// TIA Portal V19 export
FUNCTION_BLOCK "LAF_ProfinetDevDiag"   // FB73, LAD
TITLE = LAF_ProfinetDevDiag / Profinet Device Diagnose mit ProDiag
AUTHOR : Siemens Digital Industries
FAMILY : LAF
VERSION : 1.2
// The block is used for the diagnostics of the Profinet devices connected to a CPU and to display the information on the HMI. The following data will be read from the PLC and displayed via faceplates.
// * Device state 
// * Device name (max. 24 characters) 
// * Device number 
// * Group status of module errors 
// * first 8 characters of the order number (MLFB) 
// 
// The function block has to be called and configured; and the faceplates for each device have to be placed in a screen and supplied with the interface.  
// 
//  
// **PLC Data types**  
// * LAF_typeDevDiagAlarm  
// * LAF_typeDevDiagBasic  
// * LAF_typeDevDiagGlobal  
// * LAF_typeDevDiagHwAddress  
// * LAF_typeDevDiagInstruct  
// * LAF_typeDevDiagInterface  
// * LAF_typeDevDiagInternal  
// * LAF_typeDevDiagModStateMode  
// * LAF_typeDevDiagNoOfDevices  
// * LAF_typeDevDiagRisEdge  
// * LAF_typeDevDiagState  
// * LAF_typeDevDiagStateInstruct  
// * LAF_typeDevDiagStatesMode  
// * LAF_typeDevDiagStructGetDiag  
// 
// **User Constants**  
// MAX_NO_OF_MODULES  
// MAX_NO_OF_DEVICES  
// 
// 
// **WinCC Screen**  
// ![Image](LAF_ProfinetDevDiag_PrD/en/image1.PNG)
// 
// **Block call example**  
// {.pageWidth}
// ![Image]( LAF_ProfinetDevDiag_PrD/en/image42.PNG)  
// 
// **Calling interface**  
// The block must be called only once per PROFINET-IO-System in the cyclic program. The call takes place in the software unit CentralFunctions -> [CallDiagnostic](../Functions/CallDiagnostic.htm)  
// 
// **Internally used „Extended instructions / blocks“**  
// LOG2GEO, DeviceStates, GEO2LOG, ModuleStates, Get_Name, GET_IM_DATA, GET_DIAG  
// 
// **Parameters**  
// This block is provided with “pre-defined actual parameters” for structured data types, user constants, system constants etc. Therefor these parameters have to be modified only slightly or not at all, if the symbols of DBs, user constants, and system constants have not been changed.
// Die Tec-Unit diagnostiziert die an die CPU angeschlossenen Profinet Geräte um die Informationen auf dem HMI darzustellen. Folgend Daten werden gelesen und mittels eines Bildbausteins visualisiert.  
// * Geräte-Status 
// * Gerätename (max. 24 Zeichen) 
// * Geräte-Nummer 
// * Sammelzustand über Modulstörung 
// * die ersten 8 Zeichen der Bestell-/Artikelnummer (MLFB) 
// 
// Hierzu muss der Funktionsbaustein aufgerufen und parametriert werden, sowie für jedes Profinet-Gerät der vorgefertigte Bildbaustein (Faceplate) in einem Bild platziert, und mit der Schnittstelle versorgt werden.  
//  
//  
// **PLC-Datentypen**  
// 
// ![Image](LSicar_ProfinetDevDiag_PrD/de/image3.PNG)
//  
// 
// **Anwenderkonstanten**  
// MAX_NO_OF_MODULES  
// MAX_NO_OF_DEVICES  
// 
// **WinCC-Bildbaustein**  
// 
// ![Image](LSicar_ProfinetDevDiag_PrD/de/image1.PNG)
// 
// **WinCC-Bild**  
// 
// ![Image](LSicar_ProfinetDevDiag_PrD/de/image2.PNG)
// 
// **Beispielaufruf**  
// Abbildung in Kontaktplan (KOP), ohne Parameterbeschaltung. D:\Software\Symbols_Icons\BMPs-JPGs-PNGs\Verschiedene\symb_user_goto_transparent.pngEin lauffähiger Programm-Aufruf hierzu ist im „SICAR-StartUp“-Projekt enthalten.  
// 
// **Aufrufschnittstelle**  
// Der Baustein wird einmalig pro PROFINET-IO-System im zyklischen Programm aufgerufen.  
// 
// **Intern verwendete „Erweiterte Anweisungen / Bausteine“**  
// LOG2GEO, DeviceStates, GEO2LOG, ModuleStates, Get_Name, GET_IM_DATA, GET_DIAG  
// 
// **Parameter**  
// 
// ![Icon](_Icon/information.PNG)
// 
// Der Baustein ist mit "Vordefinierten Aktualparametern" versehen für Strukturvariablen, Anwender- und Systemkonstanten etc., die dadurch nicht oder nur geringfügig angepasst werden müssen, vorausgesetzt die Symbolischen Namen von DBs, Anwender-/Systemkonstanten etc. wurden nicht geändert. Die Anpassungen sind notwendig beim Index [i], z.B. für den BA-Bereich oder die HMI-/Panelnummer.  
// * Der Index ist vorbesetzt mit dem Wert [0]. Damit wird auf den Index 0 (Dummy) verwiesen. Sofern der Baustein-Parameter nicht benötigt wird, sind keine Anpassungen notwendig, andernfalls muss der Indexwert angepasst werden. 
// oder  
// * Der Index ist vorbesetzt mit [???]. Dies führt dazu, dass der Aktualparameter beim Bausteinaufruf rot markiert wird; um darauf aufmerksam zu machen, dass der Indexwert des Aktualparameters angepasst werden muss!
// stored: Access Published, IsIECCheckEnabled true, MemoryReserve 100, SetENOAutomatically true
   VAR_INPUT
      plantIdentifier { ExternalAccessible := 'False'; ExternalVisible := 'False'; ExternalWritable := 'False'} : WString[#MAX_CHAR];   // Betriebsmittel Kennzeichen. Das Kennzeichen ist auf 24 Zeichen begrenzt und sollte ein Be-triebsmittelkennzeichen, gemäß der Schaltpläne enthalten. Der Text wird im Bildbaustein, und in der Bewegungszeile ange-zeigt bzw. als Präfix für die Alarme benutzt / Identifier of the device. The identifier is limited to a length of 24 characters and should contain the name of the device according the wiring diagrams. The identifier is displayed in the faceplate and it is used as a prefix for the alarm messages.
      textListId { ExternalAccessible := 'False'; ExternalVisible := 'False'; ExternalWritable := 'False'} : Int;   // Text list ID
      localProfinetSystem { ExternalAccessible := 'False'; ExternalVisible := 'False'; ExternalWritable := 'False'} : HW_IOSYSTEM;   // Systemkonstante des lokalen „Profinet IO-Systems“. Die Variab-le befindet sich in den PLC-Variablen unter „Alle Variablen anzei-gen -> Lasche Systemkonstanten“. / System constant of the local Profinet IO system. The tag is located in PLC tags / Show all tags ->tab “System constants”.
      firstCycle { ExternalAccessible := 'False'; ExternalVisible := 'False'; ExternalWritable := 'False'} : Bool;   // Variable die den ersten CPU-Zyklus darstellt. Der Parameter ist vordefiniert und verweist auf nachfolgende Quelle. / Tag representing the first PLC cycle.
      maxDevicesDiag { ExternalAccessible := 'False'; ExternalVisible := 'False'; ExternalWritable := 'False'} : DInt;   // Maximale Anzahl von PN Devices. Der Parameter ist vordefiniert und verweist auf nachfolgende Quelle. / Maximum number of PN devices.
      maxModulesDiag { ExternalAccessible := 'False'; ExternalVisible := 'False'; ExternalWritable := 'False'} : DInt;   // Maximale Anzahl von Modulen „Der Parameter ist vordefiniert und verweist auf nachfolgende Quelle. / Maximum number of modules.
      ackAlarms { ExternalAccessible := 'False'; ExternalVisible := 'False'; ExternalWritable := 'False'} : Bool;   // Variable für Alarm quittieren. Es wird empfohlen die Variable “GlobalInterface”.globalHmi.globalAck zu verwenden. Die Varibriable wird durch den Quittier Button in der Kopfzeile versorgt. / Tag for Reset of alarms. It is recommended to use the tag “GlobalInterface”.globalHmi.globalAck” representing the Acknowledge “ACK” button in the screen header.
      hideAlarmAll { ExternalAccessible := 'False'; ExternalVisible := 'False'; ExternalWritable := 'False'} : Bool;   // Alle Störungen unterdrücken. Mit Signal TRUE werden alle Alarme unterdrückt. Hinweis: Die farbliche Animation des WinCC-Bildbausteins im PN-Diagnosebild wird immer ausgeführt. / Hide all alarms. Signal TRUE on this input, will suppress all alarms. Note: The WinCC-Faceplate in the PN-Screen will be always animated.
      hideAlarmMask { ExternalAccessible := 'False'; ExternalVisible := 'False'; ExternalWritable := 'False'} : Word;   // Einzelne Störungen unterdrücken. Bei Bedarf können einzelne Alarme deaktiviert werden, durch Setzen des entsprechenden Bits auf TRUE. Hinweis: Die farbliche Animation des WinCC-Bildbausteins im PN-Diagnosebild wird immer ausgeführt. / Hide alarm mask. Individual alarms can be suppressed by setting the corresponding bit in this mask to state TRUE (This might be necessary e.g. during commissioning). The assignment is the same as in tag “statAlarm”.
   END_VAR
   VAR_OUTPUT
      generalAlarm { ExternalAccessible := 'False'; ExternalVisible := 'False'; ExternalWritable := 'False'} : Bool;   // Sammelstörung / Group alarm.
      deviceFaulty { ExternalAccessible := 'False'; ExternalVisible := 'False'; ExternalWritable := 'False'} : Bool;   // TRUE = mindestens 1 Profinet Gerät gestört ist. / TRUE = at least one device in condition fault.
      deviceProblem { ExternalAccessible := 'False'; ExternalVisible := 'False'; ExternalWritable := 'False'} : Bool;   // TRUE = mindestens 1 Profinet Gerät ein Problem aufweist. / TRUE = at least one device with a problem.
      deviceDeactivated { ExternalAccessible := 'False'; ExternalVisible := 'False'; ExternalWritable := 'False'} : Bool;   // TRUE = mindestens 1 Profinet Gerät deaktiviert ist. / TRUE = at least one device deactivated.
      deviceNotPresent { ExternalAccessible := 'False'; ExternalVisible := 'False'; ExternalWritable := 'False'} : Bool;   // mind. 1 PN-Device nicht vorhanden, jedoch konfiguriert (z.B. ausgeschaltet) / Min. 1 device not present, but configured (e.g. switched off ).
   END_VAR
   VAR_IN_OUT
      interfaceDevDiag : "LAF_typeDevDiagInterface";   // This parameter refers to the data block "InstDevDiagInterface", which contains the information for the HMI as well as a user interface about the status of the devices. / Dieser Parameter verweist auf den Datenbaustein "DevDiagInterface“, der die Informationen für das HMI sowie eine Anwender-Schnittstelle über den Status der Devices enthält.
   END_VAR
   VAR
      statDevDiagInternal { ExternalAccessible := 'False'; ExternalVisible := 'False'; ExternalWritable := 'False'} : "LAF_typeDevDiagInternal";   // für HMI (Erreichbarkeit setzen) / for HMI (set accessebility)
      statCnt1ShotGetName { ExternalAccessible := 'False'; ExternalVisible := 'False'; ExternalWritable := 'False'} : DInt := 1;   // Einmalig "GetName": Zykluszähler PN-Devices, läuft von 1...PN_DEVDIAG_MAX-DEVICES, beginnt dann wieder bei 1 / Once only "GetName" cycle counter
      statCnt1ShotGeo2Log { ExternalAccessible := 'False'; ExternalVisible := 'False'; ExternalWritable := 'False'} : DInt := 1;   // Einmalig "GEO2LOG": Zykluszähler PN-Devices, läuft von 1...PN_DEVDIAG_MAX-DEVICES, beginnt dann wieder bei 1 / Once only "GEO2LOG" cycle counter
      statCnt1ShotGetImDat { ExternalAccessible := 'False'; ExternalVisible := 'False'; ExternalWritable := 'False'} : DInt := 1;   // Einmalig "GET_IM_DATA": Zykluszähler PN-Devices, läuft von 1...PN_DEVDIAG_MAX-DEVICES, beginnt dann wieder bei 1 / Once only "GET_IM_DATA" cycle counter
      statCntCyclDevState { ExternalAccessible := 'False'; ExternalVisible := 'False'; ExternalWritable := 'False'} : DInt := 1;   // Zyklisch für "DeviceStates": Zykluszähler PN-Devices, läuft von 1...5, beginnt dann wieder bei 1 / Cyclic "DeviceStates"cycle counter
      statCntCyclState { ExternalAccessible := 'False'; ExternalVisible := 'False'; ExternalWritable := 'False'} : DInt := 1;   // Zyklisch für "DeviceStates" rangieren in Device-Arrays: Zykluszähler PN-Devices, läuft von 1...5, beginnt dann wieder bei 1 / Cyclic "DeviceStates" cycle counter, routing to device-arrays
      statCntCyclModulState { ExternalAccessible := 'False'; ExternalVisible := 'False'; ExternalWritable := 'False'} : DInt := 1;   // Zyklisch für "ModuleStates": Zykluszähler PN-Devices, läuft von 1...PN_DEVDIAG_MAX-DEVICES, beginnt dann wieder bei 1 / Cyclic "ModuleStates" cycle counter
      statCntCyclGetDiag { ExternalAccessible := 'False'; ExternalVisible := 'False'; ExternalWritable := 'False'} : DInt := 1;   // Zyklisch für "GET_DIAG": Zykluszähler PN-Devices, läuft von 1...PN_DEVDIAG_MAX-DEVICES, beginnt dann wieder bei 1 / Cyclic "GET_DIAG" cycle counter
      statBusy { ExternalAccessible := 'False'; ExternalVisible := 'False'; ExternalWritable := 'False'} : "LAF_typeDevDiagStateInstruct";   // Busy_flags
      statDone { ExternalAccessible := 'False'; ExternalVisible := 'False'; ExternalWritable := 'False'} : "LAF_typeDevDiagStateInstruct";   // Done_flags
      statOtherInstruct { ExternalAccessible := 'False'; ExternalVisible := 'False'; ExternalWritable := 'False'} : "LAF_typeDevDiagInstruct";   // Instanzen fuer Instructions
      instGetName { ExternalAccessible := 'False'; ExternalVisible := 'False'; ExternalWritable := 'False'} : Get_Name;   // Instanzen Get_Name / Instance Get_Name
      statGetNameDat { ExternalAccessible := 'False'; ExternalVisible := 'False'; ExternalWritable := 'False'} : String[#LENGTH_GET_NAME];   // Get_Name: Name der Baugruppe / Get_Name: Name of device
      statGetNameErrorStatus { ExternalAccessible := 'False'; ExternalVisible := 'False'; ExternalWritable := 'False'} : Word;   // Get name error status
      statGetNameErrorDevCycle { ExternalAccessible := 'False'; ExternalVisible := 'False'; ExternalWritable := 'False'} : DInt;   // Zykluszähler für PN-Devices, läuft von 1...PN_DEVDIAG_MAX-DEVICES und beginnt dann wieder bei 1 usw. / Cyclic counter PN devices 1..MAX_DEVICES
      instGetImData { ExternalAccessible := 'False'; ExternalVisible := 'False'; ExternalWritable := 'False'} : Get_IM_Data;   // GET_IM_DATA
      statIm0Data { ExternalAccessible := 'False'; ExternalVisible := 'False'; ExternalWritable := 'False'} : IM0_Data;   // GET_IM_DATA
      statGetImDatErrorStatus { ExternalAccessible := 'False'; ExternalVisible := 'False'; ExternalWritable := 'False'} : Word;   // Get IM data error status
      statGetImDatErrorCycle { ExternalAccessible := 'False'; ExternalVisible := 'False'; ExternalWritable := 'False'} : DInt;   // Zykluszähler für PN-Devices, läuft von 1...PN_DEVDIAG_MAX-DEVICES und beginnt dann wieder bei 1 usw. / Cyclic counter PN devices 1..MAX_DEVICES
      statAlarm { ExternalAccessible := 'False'; ExternalVisible := 'False'; ExternalWritable := 'False'} : "LAF_typeDevDiagAlarm";   // Störungen / Alarm
      statHideAlarm { ExternalAccessible := 'False'; ExternalVisible := 'False'; ExternalWritable := 'False'} : "LAF_typeDevDiagAlarm";   // Störungen unterdrücken, Belegung identisch mit "Alarm" / Hide Alarms, identical with "Alarm"
      statRisPushbutton { ExternalAccessible := 'False'; ExternalVisible := 'False'; ExternalWritable := 'False'} : "LAF_typeDevDiagRisEdge";   // Flankenauswertung Tasten / Edge evaluation buttons
      statErrorText { ExternalAccessible := 'False'; ExternalVisible := 'False'; ExternalWritable := 'False'} : String[#LENGTH_GET_NAME] := 'No Device Name readable';   // Error text / Fehlertext
      stat8CharError { ExternalAccessible := 'False'; ExternalVisible := 'False'; ExternalWritable := 'False'} : String[#LENGTH_8_CHAR] := '????????';   // 8 character error / 8 Zeichen Fehler
      statAlarmNo { ExternalAccessible := 'False'; ExternalVisible := 'False'; ExternalWritable := 'False'} : Array[0..23] of UInt;   // Alarm Nummer für ProDiag / Alarm Number for ProDiag
   END_VAR
   VAR_TEMP
      tempDevCnt1ShotGetName : UInt;   // Type conversion / Typ Konvertierung
      tempHideAlarm : Word;   // Abbild hideAlarmMask / Image hideAlarmMask
      tempZeroWord : Word;   // Word Konstante=0 / Word constant=0
      tempZeroDword : DWord;   // DWord Konstante=0 / DWord constant=0
      tempAlarmStatus : Word;   // Abbild statAlarm / image statAlarm
   END_VAR
   VAR CONSTANT
      MAX_CHAR : DInt := 24;   // Konstante für Zeichenlänge plantidentifier / Constant length plantidentifier
      LENGTH_GET_NAME : DInt := 24;   // Length GetName / Zeichenlänge GetName
      LENGTH_8_CHAR : DInt := 8;   // Constant 8 character / Länge 8 Zeichen
   END_VAR
   // statAlarmNo[0] := 0;
   // statAlarmNo[1] := 1;
   // statAlarmNo[2] := 2;
   // statAlarmNo[3] := 3;
   // statAlarmNo[4] := 4;
   // statAlarmNo[5] := 5;
   // statAlarmNo[6] := 6;
   // statAlarmNo[7] := 7;
   // statAlarmNo[8] := 8;
   // statAlarmNo[9] := 9;
   // statAlarmNo[10] := 10;
   // statAlarmNo[11] := 11;
   // statAlarmNo[12] := 12;
   // statAlarmNo[13] := 13;
   // statAlarmNo[14] := 14;
   // statAlarmNo[15] := 15;
   // statAlarmNo[16] := 16;
   // statAlarmNo[17] := 17;
   // statAlarmNo[18] := 18;
   // statAlarmNo[19] := 19;
   // statAlarmNo[20] := 20;
   // statAlarmNo[21] := 21;
   // statAlarmNo[22] := 22;
   // statAlarmNo[23] := 23;
   VAR_TEMP   // added for the SCL form of the ladder/FBD networks
      _w1 : Bool;
      _w2 : Bool;
      _w3 : Bool;
      _w4 : Bool;
   END_VAR
BEGIN

REGION Network 1: Header Info / Änderungshistorie
   // SIEMENS AG / (c)Copyright 2024
   // ------------------------------------------------------------------------------
   // Title:            LAF_InterfaceSignalsBool
   // Comment/Function: The block is used for the diagnostics of the Profinet devices connected to a CPU and to display the information on the HMI. 
   // Library/Family:   Library of Automation Framework
   // Author:               Siemens Digital Industry
   // Tested with:      S7-PLCSIM Advanced 6.0
   // Engineering:     TIA Portal V19
   // Restrictions:      --- 
   // Requirements:  ---
   // ------------------------------------------------------------------------------
   // Change log table:
   // Version | Date | Expert in charge | Changes applied
   // -------|---------|-------------|--------------------------------------------
   // 01.02.00 | 30.09.2024 | SIMATIC Systems Support | First released version
   // Die Änderungshistorie wird nur in englischer Editiersprache geführt.
END_REGION

REGION Network 2: Description / Beschreibung
   // **Operation mode Automatic / Manual**  
   // The block is not assigned to any operation mode.  
   // 
   // **Alarms**  
   // Alarm texts are stored in the PLC alarm text lists of the software unit GlobalData. This messages are used with proDiag and also in the program alarm version of the block.  
   // 
   // | **No.** | **Message**                                                            |
   // |---------|------------------------------------------------------------------------|
   // | 1       | Invalid Value / Userconstant   "PNDevDiag": MAX_NO_OF_DEVICES [1..]     |
   // | 2       | Invalid Value / Userconstant "PNDevDiag": MAX_NO_OF_MODULES   [1..128] |
   // | 3       | Invalid Address "PNDevDiag": LOG2GEO_LOCAL_PNIO-SYSTEM                 |
   // | 4       | PROFINET Device-States: Error Read Device-States                       |
   // | 5       | PROFINET-Device faulty                                                 |
   // | 6       | PROFINET-Device with Problem                                           |
   // | 7       | Spare7                                                                 |
   // | 8       | PROFINET-Device not present but configured                             |
   // | 9       | PROFINET-Device with network error (e.g. Topology-error)               |
   // | 10      | POFINET-Device with maintenance required                               |
   // | 11      | POFINET-Device with maintenance demanded                               |
   // | 12      | Spare12                                                                |
   // | 13      | Spare13                                                                |
   // | 14      | Spare14                                                                |
   // | 15      | Spare15                                                                |
   // | 16      | Spare16                                                                |
   // | 17      | Spare17                                                                |
   // | 18      | Hide all alarm active                                                  |
   // 
   // ---
   // 
   // **User Constants**  
   // User constants are available under  the SW unit “CentralFunctions -> PLC tags -> 11_Settings -> User constants”  
   // 
   // {.pageWidth}
   // ![Image](LAF_ProfinetDevDiag_PrD/en/image4.PNG)
   // 
   // **MAX_NO_OF_DEVICES**  
   // The value of the constant should be adapted to the real number of used devices.  
   // 
   // **MAX_NO_OF_MODULES**  
   // The value of the constant should be adapted to the maximum number of used modules in a I/O station.  
   // 
   // NOTE
   // :     These values have impact on the update time of data and cycle time.  
   // 
   // ---
   // 
   // 
   // #### PLC Data types 
   // * [LAF_typeDevDiagAlarm](../Library%20Types/LAF_typeDevDiagAlarm.htm)  
   // * [LAF_typeDevDiagBasic](../Library%20Types/LAF_typeDevDiagBasic.htm)  
   // * [LAF_typeDevDiagGlobal](../Library%20Types/LAF_typeDevDiagGlobal.htm)  
   // * [LAF_typeDevDiagHwAddress](../Library%20Types/LAF_typeDevDiagHwAddress.htm)  
   // * [LAF_typeDevDiagInstruct](../Library%20Types/LAF_typeDevDiagInstruct.htm)  
   // * [LAF_typeDevDiagInterface](../Library%20Types/LAF_typeDevDiagInterface.htm)  
   // * [LAF_typeDevDiagInternal](../Library%20Types/LAF_typeDevDiagInternal.htm)  
   // * [LAF_typeDevDiagModStateMode](../Library%20Types/LAF_typeDevDiagModStateMode.htm)  
   // * [LAF_typeDevDiagNoOfDevices](../Library%20Types/LAF_typeDevDiagNoOfDevices.htm)  
   // * [LAF_typeDevDiagRisEdge](../Library%20Types/LAF_typeDevDiagRisEdge.htm)  
   // * [LAF_typeDevDiagState](../Library%20Types/LAF_typeDevDiagState.htm)  
   // * [LAF_typeDevDiagStateInstruct](../Library%20Types/LAF_typeDevDiagStateInstruct.htm)  
   // * [LAF_typeDevDiagStatesMode](../Library%20Types/LAF_typeDevDiagStatesMode.htm)  
   // * [LAF_typeDevDiagStructGetDiag](../Library%20Types/LAF_typeDevDiagStructGetDiag.htm)  
   // 
   // #### InstDevDiagInterface DB 
   // The data block “PNDevDiagInterface“is derived from the data type „LAF_typeDevDiagInterface“ and contains all information for the status to display on HMI as well as a user interface to evaluate the status program internally.  
   // {.pageWidth}
   // ![Image](LAF_ProfinetDevDiag_PrD/en/image19.PNG)
   // 
   // ---
   // 
   // **Global information**  
   // {.pageWidth}
   // ![Image](LAF_ProfinetDevDiag_PrD/en/image20.PNG)
   // 
   // ---
   // 
   // **Device status for display on HMI**  
   // {.pageWidth}
   // ![Image](LAF_ProfinetDevDiag_PrD/en/image21.PNG)
   // 
   // ---
   // 
   // **User interface device status**  
   // {.pageWidth}
   // ![Image](LAF_ProfinetDevDiag_PrD/en/image22.PNG)
   // 
   // ---
   // 
   // #### WinCC-Screen objects 
   // 
   // **WinCC Faceplate**  
   // 
   // The faceplate is available in the project library under Types -> LAF -> 10_Central -> Diagnostic -> ProfinetDevice_Diag.  
   // The faceplate consists of several WinCC objects and contains the information shown below.  
   // The faceplate is animated in terms of color depending on status and operation.   
   // 
   // {.pageWidth}
   // ![Image](LAF_ProfinetDevDiag_PrD/en/image23.PNG)
   // 
   // 
   // **WinCC Faceplate interface connection**  
   // In order to connect the faceplate with the interface tag for a Profinet device it is recommended to proceed as follows:  
   // 
   // 1. For each device, a HMI tag is available.  
   // 2. The faceplate from the project library needs to be placed in the template screen.  
   // 
   // NOTE
   // 
   // :     The data interface is available in data block „InstDevDiagInterface“.  
   // :     The array index number corresponds with the device number.  
   // :     Index [0] are not used.  
   // :     The tag has to be assigned to Properties -> Interface -> HMI.
   // 
   // ---
   // 
   // **WinCC Screen template for placement of the faceplates**  
   // The faceplate is available in the project navigation under Screens -> 09_Diagnostics -> 53_PnDiagnostic.  
   // The screen consists of several WinCC objects and contains the shown below information.  
   // 
   // {.pageWidth}
   // ![Image](LAF_ProfinetDevDiag_PrD/en/image40.PNG)
   // 
   // 
   // #### Further information 
   // 
   // #### Update info 
   //  
   // #### Further documentation
   // **Betriebsart Automatik / Hand**  
   // Der Baustein ist keiner Betriebsart / Betriebsartenbereich zugeordnet.  
   // 
   // **Alarme**  
   // Anstehende Alarme können über die OUTPUT-Parameter für den weiteren Programmablauf verwendet werden.  Alarme können über den „QUIT“-Button im HMI-Bild quittiert werden.  
   // 
   // **Alarm**  
   // Die statische Strukturvariable „statAlarm“ hat folgende Belegung:  
   // 
   // |       statAlarm. [Word]  |  |  |
   // |---|---|---|
   // |     Bitposition  |   Bezeichnung  |   Erläuterung  |
   // |     %X0  |   #.invalidValueMaxDevices  |   Input kleiner/gleich angegeben, muss grösser/gleich 1 sein [1..]  |
   // |     %X1  |   #.invalidValueMaxModules  |   Input kleiner/gleich 0 oder grösser angegeben, gültig [1..128]  |
   // |     %X2  |   #.InvalidAddressLog2Geo  |   ungültige Adresse an LADDR bei LOG2GEO bzw. an Input  |
   // |     %X3  |   #.errorReadDeviceState  |   Fehler beim Lesen der Baugruppenzustandsinformationen  |
   // |     %X4  |   #.deviceFaulty  |   mind. 1 PN-Device gestört  |
   // |     %X5  |   #.deviceProblem  |   mind. 1 PN-Device hat ein Problem  |
   // |     %X6  |   #.deviceDeactivated  |   mind. 1 PN-Device deaktiviert -Dies ist kein Fehler, lediglich in Struktur gelistet-  |
   // |     %X7  |   #.deviceNotPresent  |   mind. 1 PN-Device nicht vorhanden, jedoch konfiguriert (z.B. konfiguriert und ausgeschaltet)  |
   // |     %X8  |   #.deviceNetworkError  |   mind. 1 PN-Device mit Netzwerkfehler (z.B. Topologie-Fehler)  |
   // |     %X9  |   #.deviceMaintRequired  |   mind. 1 PN-Device mit Wartungsbedarf  |
   // |     %X10  |   #.deviceMaintDemanded  |   mind. 1 PN-Device mit Wartungsanforderung  |
   // |     %X11 .. 15  |   #.spare..  |   Reserve  |
   // 
   // 
   // **Anwenderkonstanten**  
   // Anwenderkonstanten verfügbar unter PLC-Variablen/Alle Variablen anzeigen -> Anwenderkonstanten.  
   // 
   // {.pageWidth}
   // ![Image](LSicar_ProfinetDevDiag_PrD/de/image4.PNG)
   // 
   // **MAX_NO_OF_DEVICES**  
   // Die Anwenderkonstante sollte, auf die auf die tatsächlichen Anzahl Geräte angepasst werden.  
   // 
   // **MAX_NO_OF_MODULES**  
   // Die Anwenderkonstante sollte, auf die auf die maximale Anzahl Module angepasst werden.  
   // 
   // NOTE
   // :     In Abhängigkeit von dem Wert der Variablen hängt die Aktualisierungszeit der Daten und auch somit auch die Zykluszeit.
   // 
   // ---
   // 
   // #### PLC-Datentypen
   // 
   // Verwendete PLC-Datentypen für den SPS-Programmbaustein / WinCC-Bildbaustein/Faceplate:  
   // 
   // **LSicar_typeDevDiagAlarm**  
   // Dieser PLC-Datentyp beinhaltet die Struktur der möglichen Alarme  
   // 
   // {.pageWidth}
   // ![Image](LSicar_ProfinetDevDiag_PrD/de/image5.PNG)
   //  
   // 
   // **_typeDevDiagBasic**  
   // Dieser PLC-Datentyp beinhaltet die Informationen für den Bildbaustein   
   // 
   // {.pageWidth}
   // ![Image](LSicar_ProfinetDevDiag_PrD/de/image6.PNG)
   // 
   // 
   // **_typeDevDiagGlobal**  
   // Dieser PLC-Datentyp beinhaltet globale Daten, für das HMI-Popup.   
   // 
   // {.pageWidth}
   // ![Image](LSicar_ProfinetDevDiag_PrD/de/image7.PNG) 
   // 
   // 
   // **_typeDevDiagHwAddress**  
   // Dieser PLC-Datentyp beinhaltet Informationen der auszuwertenden HW Typen.  
   // 
   // {.pageWidth}
   // ![Image](LSicar_ProfinetDevDiag_PrD/de/image8.PNG) 
   // 
   // **_typeDevDiagInstruct**  
   // Dieser PLC-Datentyp beinhaltet die Struktur der ausgelesen Diagnose Daten  
   // 
   // {.pageWidth}
   // ![Image](LSicar_ProfinetDevDiag_PrD/de/image9.PNG)
   // 
   // **_typeDevDiagInterface**  
   // Dieser PLC-Datentyp bildet die Struktur für den Datenbaustein „DevDiagInterface“.    
   // 
   // {.pageWidth}
   // ![Image](LSicar_ProfinetDevDiag_PrD/de/image10.PNG) 
   // 
   // **_typeDevDiagInternal**  
   // Dieser PLC-Datentyp beinhaltet interne Daten für die Bearbeitung des Funktionsbausteines, die nicht am HMI angezeigt werden.  
   // 
   // {.pageWidth}
   // ![Image](LSicar_ProfinetDevDiag_PrD/de/image11.PNG) 
   // 
   // **_typeDevDiagModStateMode**  
   // Dieser PLC-Datentyp beinhaltet die Struktur der Parameter sowie die Rückgabewerte der Module.  
   // 
   // {.pageWidth}
   // ![Image](LSicar_ProfinetDevDiag_PrD/de/image12.PNG)
   // 
   // **_typeDevDiagNoOfDevices**  
   // Dieser PLC-Datentyp beinhaltet die Anzahl der Geräte, die diesen Status-Informationen entsprechen.  
   // 
   // {.pageWidth}
   // ![Image](LSicar_ProfinetDevDiag_PrD/de/image13.PNG)
   // 
   // **_typeDevDiagRisEdge**
   // Dieser PLC-Datentyp beinhaltet die Struktur für Flanken-Auswertungen  
   // 
   // {.pageWidth}
   // ![Image](LSicar_ProfinetDevDiag_PrD/de/image14.PNG)
   // 
   // **_typeDevDiagState**  
   // Dieser PLC Datentyp beinhaltet die Status Informationen der Geräte und dient als Anwender-Schnittstelle.   
   // 
   // {.pageWidth}
   // ![Image](LSicar_ProfinetDevDiag_PrD/de/image15.PNG)
   // 
   // **_typeDevDiagStateInstruct**  
   // Dieser PLC-Datentyp beinhaltet die Status Informationen der laufenden Anweisungen.  
   // 
   // {.pageWidth}
   // ![Image](LSicar_ProfinetDevDiag_PrD/de/image16.PNG)
   //  
   // **_typeDevDiagStatesMode**  
   // Dieser PLC-Datentyp beinhaltet die Struktur der Parameter sowie die Rückgabewerte der Geräte.  
   // 
   // {.pageWidth}
   // ![Image](LSicar_ProfinetDevDiag_PrD/de/image17.PNG)
   // 
   // **_typeDevDiagStructGetDiag**  
   // Dieser PLC-Datentyp beinhaltet die Struktur der Anweisung GETDIAG  
   // 
   // {.pageWidth}
   // ![Image](LSicar_ProfinetDevDiag_PrD/de/image18.PNG)
   //  
   // 
   // #### DevDiagInterface DB 
   // Der Datenbaustein „DevDiagInterface“ ist abgeleitet vom PLC Datentyp „LSicar_typeDevDiagInterface“ und beinhaltet sowohl alle Informationen zur Status-Anzeige im HMI als auch eine Anwender-Schnittstelle zur Auswertung des Status für programminterne Zwecke.  
   // 
   // {.pageWidth}
   // ![Image](LSicar_ProfinetDevDiag_PrD/de/image19.PNG)
   // 
   // Global information  
   // 
   // {.pageWidth}
   // ![Image](LSicar_ProfinetDevDiag_PrD/de/image20.PNG)
   // 
   //  
   // Device Status zur Anzeige am HMI  
   // 
   // {.pageWidth}
   // ![Image](LSicar_ProfinetDevDiag_PrD/de/image21.PNG)
   // 
   // Anwender-Schnittstelle Device Status  
   // 
   // {.pageWidth}
   // ![Image](LSicar_ProfinetDevDiag_PrD/de/image22.PNG)
   // 
   // 
   // #### WinCC Bildobjekte 
   // 
   // **WinCC-Bildbaustein**  
   // Der Bildbaustein befindet sich in der Projekt-Bibliothek unter „Typen“.  
   // Der Bildbaustein ist erstellt aus mehreren einzelnen WinCC-Objekten und enthält die dargestellten Informationen. Der Bildbaustein wird farblich animiert, je nach Zustand und Bewegung. Durch Klick auf den Bildbaustein wird in das dazugehörige WinCC (Diagnose) Bild verzweigt, sofern in „Eigenschaften -> Ereignisse“ die entsprechenden Ereignisse projekteirt sind.  
   // 
   // {.pageWidth}
   // ![Image](LSicar_ProfinetDevDiag_PrD/de/image23.PNG)
   // 
   // **Farbgebung / Animation des Bildbausteins (Faceplate)**    
   //  
   //  |       Objekt / Farbe |  |     Bedeutung / Farbe   |
   // |---|---|:---:|
   // |     Profinet Gerätename und Farbanimation  |  |  |
   // |     Gerätename  |   Es wird der in der Hardware-Konfiguration angegeben Gerätename ausgelesen und angezeigt (max. 24 Zeichen).  |  |
   // |     ![Image](LSicar_ProfinetDevDiag_PrD/de/image25.PNG)   |   Gerät ist konfiguriert, vorhanden, aktiviert und fehlerfrei  |  |
   // |     ![Image](LSicar_ProfinetDevDiag_PrD/de/image26.PNG)   |   Gerät ist konfiguriert, aber nicht vorhanden   |  |
   // |     ![Image](LSicar_ProfinetDevDiag_PrD/de/image27.PNG)   |   Gerät ist deaktiviert   |  |
   // |     ![Image](LSicar_ProfinetDevDiag_PrD/de/image28.PNG)   |   Gerät ist gestört   |  |
   // |     ![Image](LSicar_ProfinetDevDiag_PrD/de/image29.PNG)   |   Gerät war gestört   |  |
   // |     ![Image](LSicar_ProfinetDevDiag_PrD/de/image30.PNG)   |   Gerät hat ein Problem   |  |
   // |     ![Image](LSicar_ProfinetDevDiag_PrD/de/image31.PNG)   |   Gerät hatte ein Problem   |  |
   // |     ![Image](LSicar_ProfinetDevDiag_PrD/de/image32.PNG)   |  Kann der Gerätename kann nicht gelesen werden, so wird der Text „No Device Name readable!“ angezeigt. Dies ist ein Hinweis darauf, dass das Gerät möglicherweise nicht konfiguriert und/oder vorhanden ist.   |  |
   // |     Netzsymbol  |  |  |
   // |       ![Image](LSicar_ProfinetDevDiag_PrD/de/image33.PNG)  |  Netzwerk Fehler von Gerät 
   //  - Grün: kein Fehler 
   //  - Rot: Fehler (z.B. Topologiefehler)   |  |
   // |     Gerätenummer  |  |  |
   // |     Beispiel: 25   |   Hier wird die Gerätenummer des Gerätes angezeigt.  |  |
   // |     Modulfehler / Wartung  |  |  |
   // |     ![Image](LSicar_ProfinetDevDiag_PrD/de/image34.PNG)   |   Symbol: Modulfehler  |  |
   // |     ![Image](LSicar_ProfinetDevDiag_PrD/de/image35.PNG)   |   Symbol: Wartungsbedarf  |  |
   // |     ![Image](LSicar_ProfinetDevDiag_PrD/de/image36.PNG)   |   Symbol: Wartungsanforderung  |  |
   // |     Tec-Unit Type  |  |  |
   // |     ![Image](LSicar_ProfinetDevDiag_PrD/de/image37.PNG)   |   Name des Tec-Unit Typs  |  |
   // |     Artikel Bestellnummer (MLFB)  |  |  |
   // |     Beispiel: ![Image](LSicar_ProfinetDevDiag_PrD/de/image38.PNG)   |   Hier werden die ersten 8 Zeichen der Artikel-/Bestellnummer (MLFB) dargestellt. Kann diese Information nicht gelesen werden, so werden ‘????????‘ angezeigt. Dies ist ein Hinweis darauf, dass das Gerät möglicherweise nicht konfiguriert und/oder nicht vorhanden ist.    |  |
   // 
   // 
   // **WinCC-Bildbaustein - Schnittstellenversorgung**  
   // Um den Bildbaustein (Faceplate) für ein Profinet-Gerät mit den notwendigen Daten zu versorgen, gehen Sie wie folgt vor.  
   // 
   // 1. Für jedes PN-Gerät ist eine HMI-Variable angelegt.  
   // 2. Der Bildbaustein aus der Projekt Bibliothek wird in dem Bild platziert. Die Variable muss unter „Eigenschaften -> Schnittstelle“. dem Bildbaustein zugewiesen werden.  
   //   
   // {.pageWidth}
   // ![Image](LSicar_ProfinetDevDiag_PrD/de/image39.PNG)
   // 
   // NOTE
   // :     Die Daten hierzu sind im Datenbaustein „DevDiagInterface“ hinterlegt.  
   // :     Die Index Nummer entspricht der Geräte Nummer. 
   // :     Index [0] wird nicht verwendet. 
   // 
   // ---
   // 
   // **WinCC-Bildvorlage, zur Platzierung der Bildbausteine**  
   // Das Bild befindet sich im Projekt (Projektnavigation) im HMI-Teil unter „Bilder“.  
   // Es ist erstellt aus mehreren einzelnen WinCC-Objekten und enthält die dargestellten Informationen.  
   // 
   // {.pageWidth}
   // ![Image](LSicar_ProfinetDevDiag_PrD/de/image40.PNG)
   // 
   // #### Beispiel 
   // Die Bildbausteine/ Faceplates für die Profinet Geräte Diagnose werden innerhalb eines Bildes platziert und mit der zugehörigen HMI-Variablen verbunden.  
   // Im Beispiel- Bild (rechts) werden die Informationen zur Verfügung gestellt.  
   // 
   // {.pageWidth}
   // ![Image](LSicar_ProfinetDevDiag_PrD/de/image41.PNG)
   // 
   // 
   // #### FWeitere Hinweise
   // 
   // #### Updateinfo 
   //  
   // #### Weitere Dokumente 
   // 
   // ![Icon](_Icon/reference.PNG)
   // 
   // Siehe ..\SICAR_Global\SICAR_Tec-Unit_HMI-Objects.pdf
END_REGION

REGION Network 3: Initialize / Initialisieren
   // Initialization of the values / Initialisieren der Werte
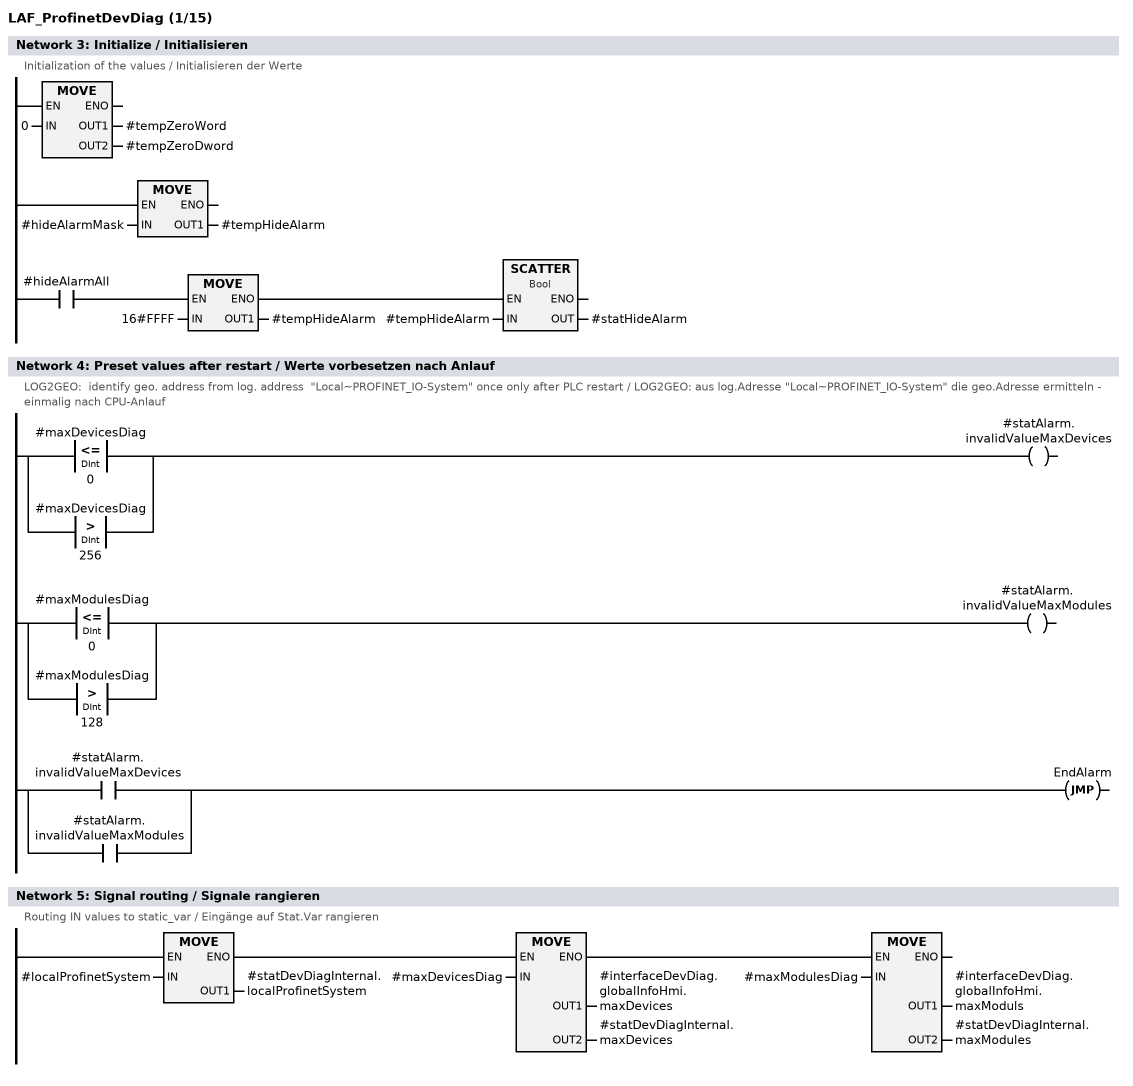
   RUNG wire#powerrail
      Move(in := 0, out1 => #tempZeroWord, out2 => #tempZeroDword)
   END_RUNG
   RUNG wire#powerrail
      Move(in := #hideAlarmMask, out1 => #tempHideAlarm)
   END_RUNG
   RUNG wire#powerrail
      Contact( #hideAlarmAll )
      Move(in := 16#FFFF, out1 => #tempHideAlarm)
      { S7_Templates := "[dest_type := Bool, src_type := Word]" } SCATTER(IN := #tempHideAlarm, OUT => #statHideAlarm)
   END_RUNG
   // the same network as SCL:
   #tempZeroWord := 0;
   #tempZeroDword := 0;
   #tempHideAlarm := #hideAlarmMask;
   IF #hideAlarmAll THEN
       #tempHideAlarm := 16#FFFF;
       SCATTER(IN := #tempHideAlarm, OUT => #statHideAlarm);
   END_IF;
END_REGION

REGION Network 4: Preset values after restart / Werte vorbesetzen nach Anlauf
   // LOG2GEO:  identify geo. address from log. address  "Local~PROFINET_IO-System" once only after PLC restart / LOG2GEO: aus log.Adresse "Local~PROFINET_IO-System" die geo.Adresse ermitteln - einmalig nach CPU-Anlauf
   RUNG wire#powerrail
      { S7_Templates := "SrcType := DInt" } LE_Contact(in1 := #maxDevicesDiag, in2 := 0)
      wire#w1
      Coil( #statAlarm.invalidValueMaxDevices )
   END_RUNG
   RUNG wire#powerrail
      { S7_Templates := "SrcType := DInt" } GT_Contact(in1 := #maxDevicesDiag, in2 := 256)
   END_RUNG wire#w1
   RUNG wire#powerrail
      { S7_Templates := "SrcType := DInt" } LE_Contact(in1 := #maxModulesDiag, in2 := 0)
      wire#w2
      Coil( #statAlarm.invalidValueMaxModules )
   END_RUNG
   RUNG wire#powerrail
      { S7_Templates := "SrcType := DInt" } GT_Contact(in1 := #maxModulesDiag, in2 := 128)
   END_RUNG wire#w2
   RUNG wire#powerrail
      Contact( #statAlarm.invalidValueMaxDevices )
      wire#w3
      JumpCoil( EndAlarm )
   END_RUNG
   RUNG wire#powerrail
      Contact( #statAlarm.invalidValueMaxModules )
   END_RUNG wire#w3
   // the same network as SCL:
   #statAlarm.invalidValueMaxDevices := (#maxDevicesDiag <= 0) OR (#maxDevicesDiag > 256);
   #statAlarm.invalidValueMaxModules := (#maxModulesDiag <= 0) OR (#maxModulesDiag > 128);
   IF #statAlarm.invalidValueMaxDevices OR #statAlarm.invalidValueMaxModules THEN GOTO EndAlarm; END_IF;
END_REGION

REGION Network 5: Signal routing / Signale rangieren
   // Routing IN values to static_var / Eingänge auf Stat.Var rangieren
   RUNG wire#powerrail
      Move(in := #localProfinetSystem, out1 => #statDevDiagInternal.localProfinetSystem)
      Move(in := #maxDevicesDiag, out1 => #interfaceDevDiag.globalInfoHmi.maxDevices, out2 => #statDevDiagInternal.maxDevices)
      Move(in := #maxModulesDiag, out1 => #interfaceDevDiag.globalInfoHmi.maxModuls, out2 => #statDevDiagInternal.maxModules)
   END_RUNG
   // the same network as SCL:
   #statDevDiagInternal.localProfinetSystem := #localProfinetSystem;
   #interfaceDevDiag.globalInfoHmi.maxDevices := #maxDevicesDiag;
   #statDevDiagInternal.maxDevices := #maxDevicesDiag;
   #interfaceDevDiag.globalInfoHmi.maxModuls := #maxModulesDiag;
   #statDevDiagInternal.maxModules := #maxModulesDiag;
END_REGION

REGION Network 6: Initialization / Initialisierung
   // Init after restart PLC or manual request / Initialisierung nach CPU Anlauf
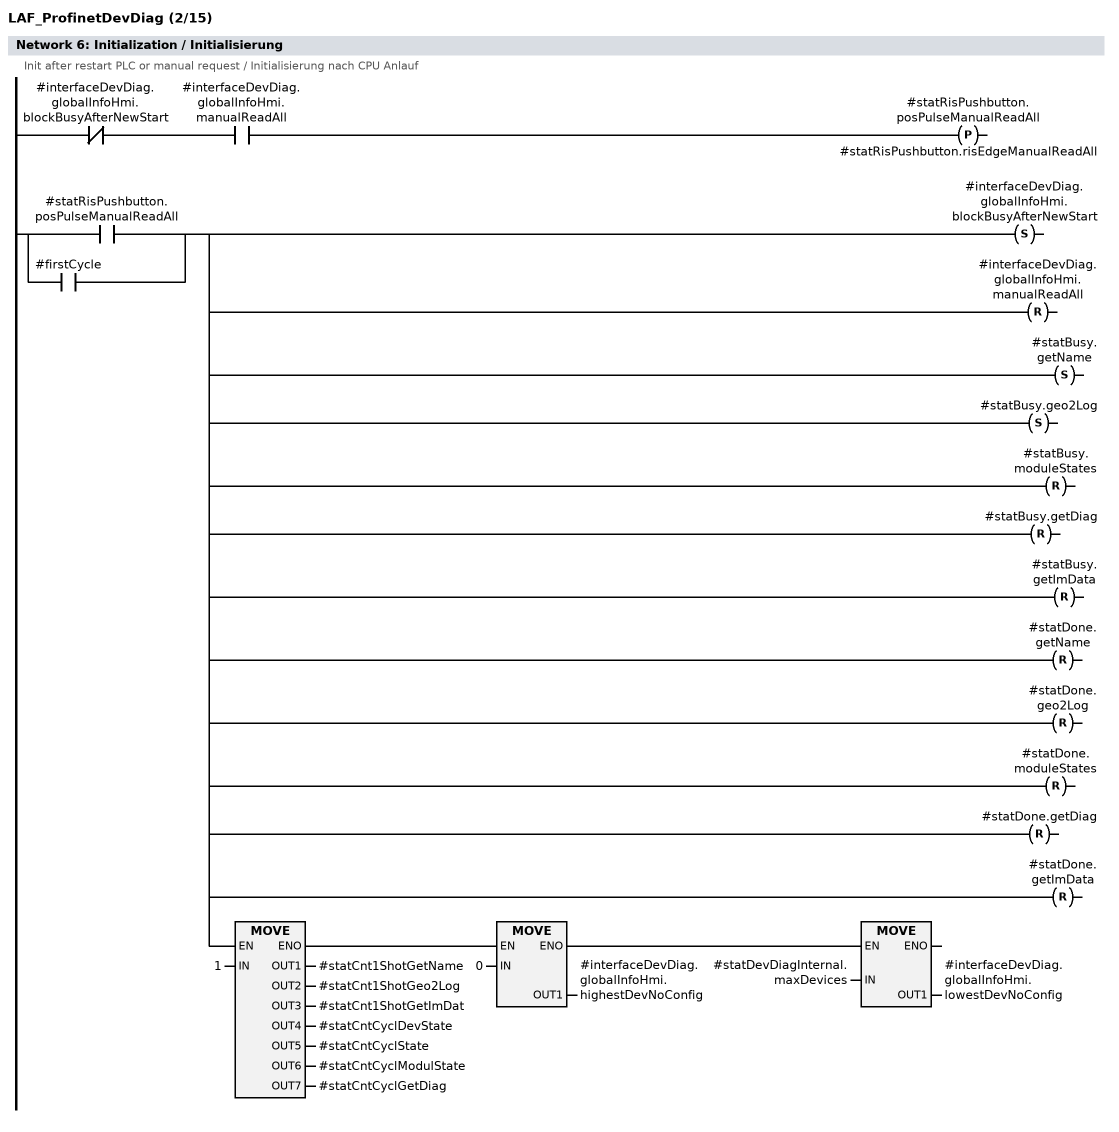
   #_w1 := NOT #interfaceDevDiag.globalInfoHmi.blockBusyAfterNewStart AND #interfaceDevDiag.globalInfoHmi.manualReadAll;
   #statRisPushbutton.posPulseManualReadAll := #_w1 AND NOT #statRisPushbutton.risEdgeManualReadAll;   // rising edge
   #statRisPushbutton.risEdgeManualReadAll := #_w1;
   IF #statRisPushbutton.posPulseManualReadAll OR #firstCycle THEN
       #interfaceDevDiag.globalInfoHmi.blockBusyAfterNewStart := TRUE;
       #interfaceDevDiag.globalInfoHmi.manualReadAll := FALSE;
       #statBusy.getName := TRUE;
       #statBusy.geo2Log := TRUE;
       #statBusy.moduleStates := FALSE;
       #statBusy.getDiag := FALSE;
       #statBusy.getImData := FALSE;
       #statDone.getName := FALSE;
       #statDone.geo2Log := FALSE;
       #statDone.moduleStates := FALSE;
       #statDone.getDiag := FALSE;
       #statDone.getImData := FALSE;
       #statCnt1ShotGetName := 1;
       #statCnt1ShotGeo2Log := 1;
       #statCnt1ShotGetImDat := 1;
       #statCntCyclDevState := 1;
       #statCntCyclState := 1;
       #statCntCyclModulState := 1;
       #statCntCyclGetDiag := 1;
       #interfaceDevDiag.globalInfoHmi.highestDevNoConfig := 0;
       #interfaceDevDiag.globalInfoHmi.lowestDevNoConfig := #statDevDiagInternal.maxDevices;
   END_IF;
END_REGION

REGION Network 7: Read slot number of HW / Lesen der Slotnummer der HW
   // Once only read "LOG2GEO" after restart PLC or manual request, to get the slot number of the HW ID. / Einmailges Lesen LOG2GEO: nach CPU-Neustart oder man. Leseanstoß HMI, um die Slotnummer der HW ID zu erhalten
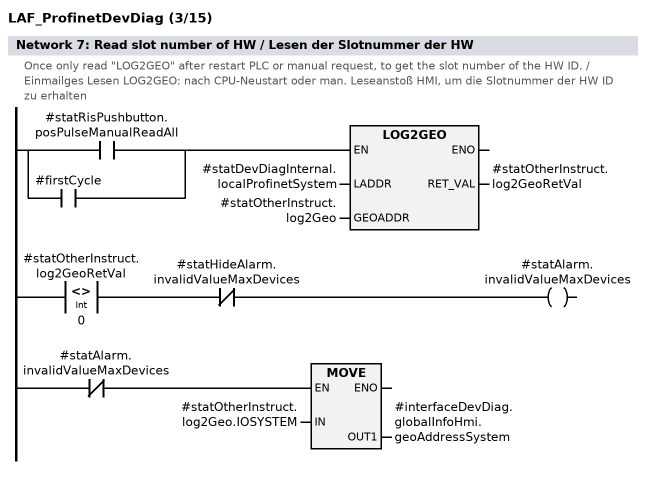
   RUNG wire#powerrail
      Contact( #statRisPushbutton.posPulseManualReadAll )
      wire#w1
      LOG2GEO(LADDR := #statDevDiagInternal.localProfinetSystem, GEOADDR := #statOtherInstruct.log2Geo, Ret_Val => #statOtherInstruct.log2GeoRetVal)
   END_RUNG
   RUNG wire#powerrail
      Contact( #firstCycle )
   END_RUNG wire#w1
   RUNG wire#powerrail
      { S7_Templates := "SrcType := Int" } NE_Contact(in1 := #statOtherInstruct.log2GeoRetVal, in2 := 0)
      I_Contact( #statHideAlarm.invalidValueMaxDevices )
      Coil( #statAlarm.invalidValueMaxDevices )
   END_RUNG
   RUNG wire#powerrail
      I_Contact( #statAlarm.invalidValueMaxDevices )
      Move(in := #statOtherInstruct.log2Geo.IOSYSTEM, out1 => #interfaceDevDiag.globalInfoHmi.geoAddressSystem)
   END_RUNG
   // the same network as SCL:
   IF #statRisPushbutton.posPulseManualReadAll OR #firstCycle THEN
       #statOtherInstruct.log2GeoRetVal := LOG2GEO(LADDR := #statDevDiagInternal.localProfinetSystem,
                               GEOADDR := #statOtherInstruct.log2Geo);
   END_IF;
   #statAlarm.invalidValueMaxDevices := (#statOtherInstruct.log2GeoRetVal <> 0) AND NOT #statHideAlarm.invalidValueMaxDevices;
   IF NOT #statAlarm.invalidValueMaxDevices THEN
       #interfaceDevDiag.globalInfoHmi.geoAddressSystem := #statOtherInstruct.log2Geo.IOSYSTEM;
   END_IF;
END_REGION

REGION Network 8: ResetHistoryAll_HMI
   // Reset of the whole history data / Reseten aller historischer Daten
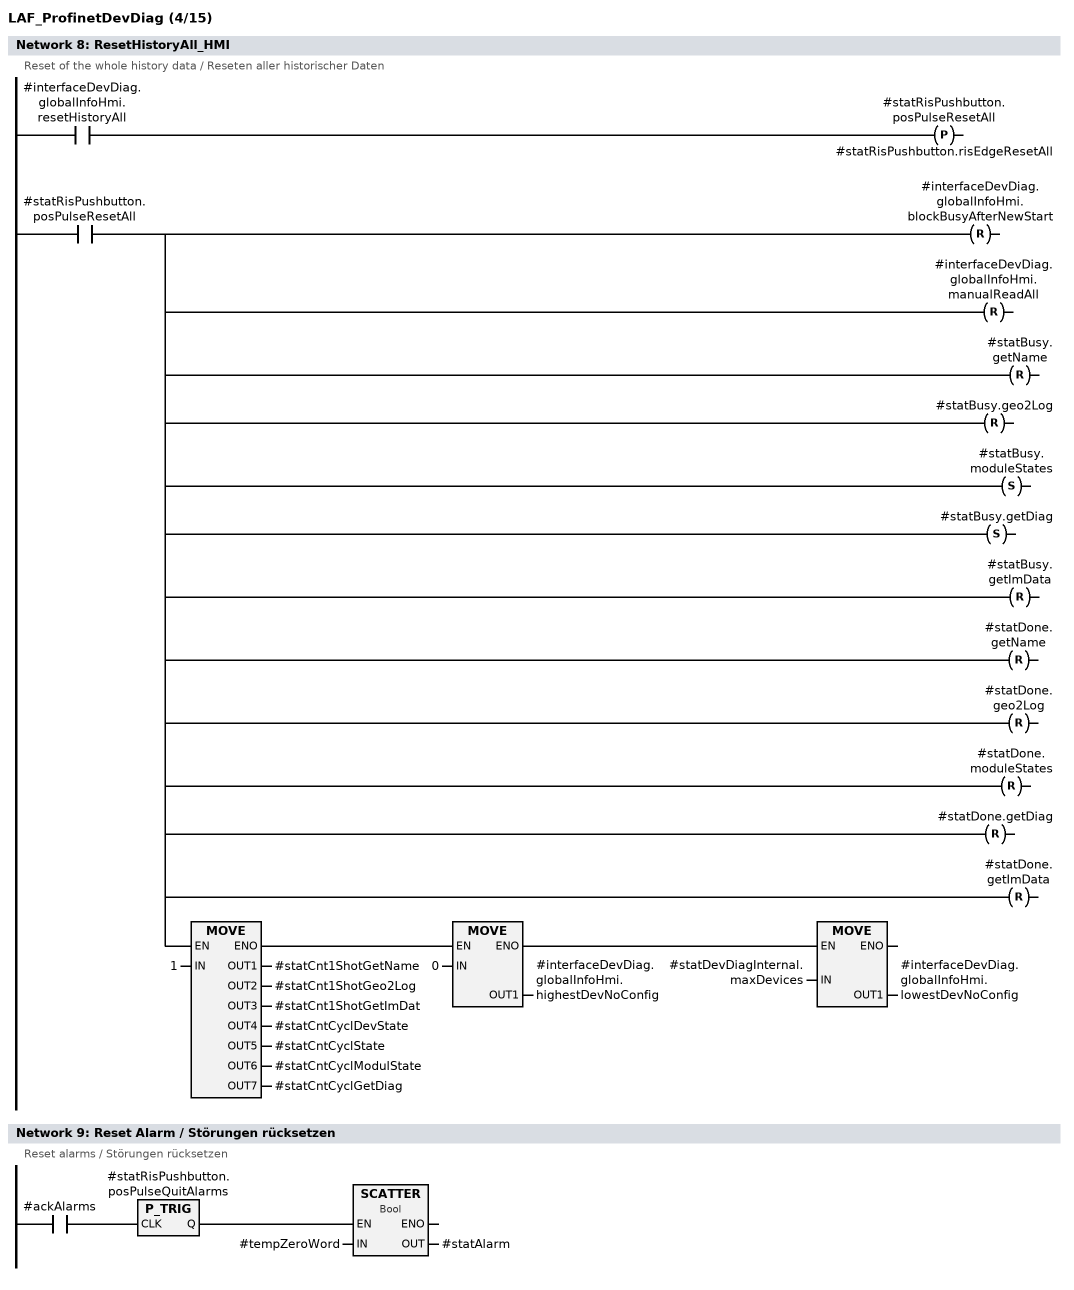
   #statRisPushbutton.posPulseResetAll := #interfaceDevDiag.globalInfoHmi.resetHistoryAll AND NOT #statRisPushbutton.risEdgeResetAll;   // rising edge
   #statRisPushbutton.risEdgeResetAll := #interfaceDevDiag.globalInfoHmi.resetHistoryAll;
   IF #statRisPushbutton.posPulseResetAll THEN
       #interfaceDevDiag.globalInfoHmi.blockBusyAfterNewStart := FALSE;
       #interfaceDevDiag.globalInfoHmi.manualReadAll := FALSE;
       #statBusy.getName := FALSE;
       #statBusy.geo2Log := FALSE;
       #statBusy.moduleStates := TRUE;
       #statBusy.getDiag := TRUE;
       #statBusy.getImData := FALSE;
       #statDone.getName := FALSE;
       #statDone.geo2Log := FALSE;
       #statDone.moduleStates := FALSE;
       #statDone.getDiag := FALSE;
       #statDone.getImData := FALSE;
       #statCnt1ShotGetName := 1;
       #statCnt1ShotGeo2Log := 1;
       #statCnt1ShotGetImDat := 1;
       #statCntCyclDevState := 1;
       #statCntCyclState := 1;
       #statCntCyclModulState := 1;
       #statCntCyclGetDiag := 1;
       #interfaceDevDiag.globalInfoHmi.highestDevNoConfig := 0;
       #interfaceDevDiag.globalInfoHmi.lowestDevNoConfig := #statDevDiagInternal.maxDevices;
   END_IF;
END_REGION

REGION Network 9: Reset Alarm / Störungen rücksetzen
   // Reset alarms / Störungen rücksetzen
   RUNG wire#powerrail
      Contact( #ackAlarms )
      P_Trig( #statRisPushbutton.posPulseQuitAlarms )
      { S7_Templates := "[dest_type := Bool, src_type := Word]" } SCATTER(IN := #tempZeroWord, OUT => #statAlarm)
   END_RUNG
   // the same network as SCL:
   #_w1 := #ackAlarms AND NOT #statRisPushbutton.posPulseQuitAlarms;   // rising edge
   #statRisPushbutton.posPulseQuitAlarms := #ackAlarms;
   IF #_w1 THEN SCATTER(IN := #tempZeroWord, OUT => #statAlarm); END_IF;
END_REGION

REGION Network 10: Read Device State Mode 1..5 / DeviceStates: Aufruf - Zustände und Anzahl der PN-Devices ermitteln
   // Read the device state. Only once per cycle / Lesen des Gerätezustands. Nur ein Gerät pro Programmzyklus
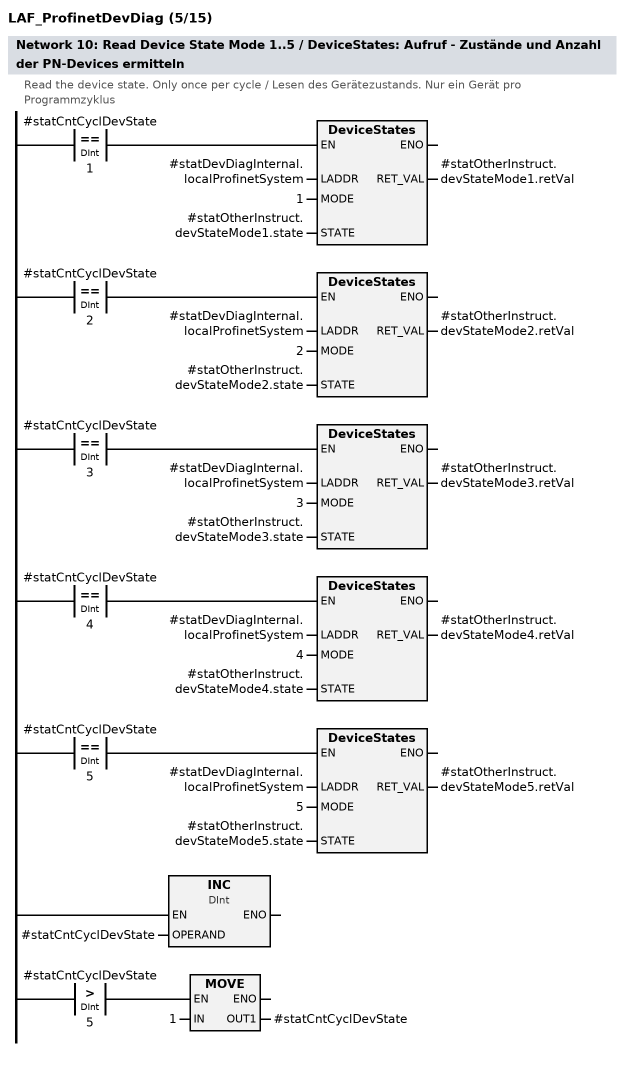
   RUNG wire#powerrail
      { S7_Templates := "SrcType := DInt" } EQ_Contact(in1 := #statCntCyclDevState, in2 := 1)
      DeviceStates(LADDR := #statDevDiagInternal.localProfinetSystem, MODE := 1, STATE := #statOtherInstruct.devStateMode1.state, Ret_Val => #statOtherInstruct.devStateMode1.retVal)
   END_RUNG
   RUNG wire#powerrail
      { S7_Templates := "SrcType := DInt" } EQ_Contact(in1 := #statCntCyclDevState, in2 := 2)
      DeviceStates(LADDR := #statDevDiagInternal.localProfinetSystem, MODE := 2, STATE := #statOtherInstruct.devStateMode2.state, Ret_Val => #statOtherInstruct.devStateMode2.retVal)
   END_RUNG
   RUNG wire#powerrail
      { S7_Templates := "SrcType := DInt" } EQ_Contact(in1 := #statCntCyclDevState, in2 := 3)
      DeviceStates(LADDR := #statDevDiagInternal.localProfinetSystem, MODE := 3, STATE := #statOtherInstruct.devStateMode3.state, Ret_Val => #statOtherInstruct.devStateMode3.retVal)
   END_RUNG
   RUNG wire#powerrail
      { S7_Templates := "SrcType := DInt" } EQ_Contact(in1 := #statCntCyclDevState, in2 := 4)
      DeviceStates(LADDR := #statDevDiagInternal.localProfinetSystem, MODE := 4, STATE := #statOtherInstruct.devStateMode4.state, Ret_Val => #statOtherInstruct.devStateMode4.retVal)
   END_RUNG
   RUNG wire#powerrail
      { S7_Templates := "SrcType := DInt" } EQ_Contact(in1 := #statCntCyclDevState, in2 := 5)
      DeviceStates(LADDR := #statDevDiagInternal.localProfinetSystem, MODE := 5, STATE := #statOtherInstruct.devStateMode5.state, Ret_Val => #statOtherInstruct.devStateMode5.retVal)
   END_RUNG
   RUNG wire#powerrail
      { S7_Templates := "DestType := DInt" } Inc( #statCntCyclDevState )
   END_RUNG
   RUNG wire#powerrail
      { S7_Templates := "SrcType := DInt" } GT_Contact(in1 := #statCntCyclDevState, in2 := 5)
      Move(in := 1, out1 => #statCntCyclDevState)
   END_RUNG
   // the same network as SCL:
   IF #statCntCyclDevState = 1 THEN
       #statOtherInstruct.devStateMode1.retVal := DeviceStates(LADDR := #statDevDiagInternal.localProfinetSystem,
                               MODE := 1,
                               STATE := #statOtherInstruct.devStateMode1.state);
   END_IF;
   IF #statCntCyclDevState = 2 THEN
       #statOtherInstruct.devStateMode2.retVal := DeviceStates(LADDR := #statDevDiagInternal.localProfinetSystem,
                               MODE := 2,
                               STATE := #statOtherInstruct.devStateMode2.state);
   END_IF;
   IF #statCntCyclDevState = 3 THEN
       #statOtherInstruct.devStateMode3.retVal := DeviceStates(LADDR := #statDevDiagInternal.localProfinetSystem,
                               MODE := 3,
                               STATE := #statOtherInstruct.devStateMode3.state);
   END_IF;
   IF #statCntCyclDevState = 4 THEN
       #statOtherInstruct.devStateMode4.retVal := DeviceStates(LADDR := #statDevDiagInternal.localProfinetSystem,
                               MODE := 4,
                               STATE := #statOtherInstruct.devStateMode4.state);
   END_IF;
   IF #statCntCyclDevState = 5 THEN
       #statOtherInstruct.devStateMode5.retVal := DeviceStates(LADDR := #statDevDiagInternal.localProfinetSystem,
                               MODE := 5,
                               STATE := #statOtherInstruct.devStateMode5.state);
   END_IF;
   #statCntCyclDevState := #statCntCyclDevState + 1;
   IF #statCntCyclDevState > 5 THEN #statCntCyclDevState := 1; END_IF;
END_REGION

REGION Network 11: Evaluate "Ret_Val" / Auswertung "Ret_Val"
   // Evaluate  "Ret_Value"  for read error. / Fehlerauswertung für Ret_Value
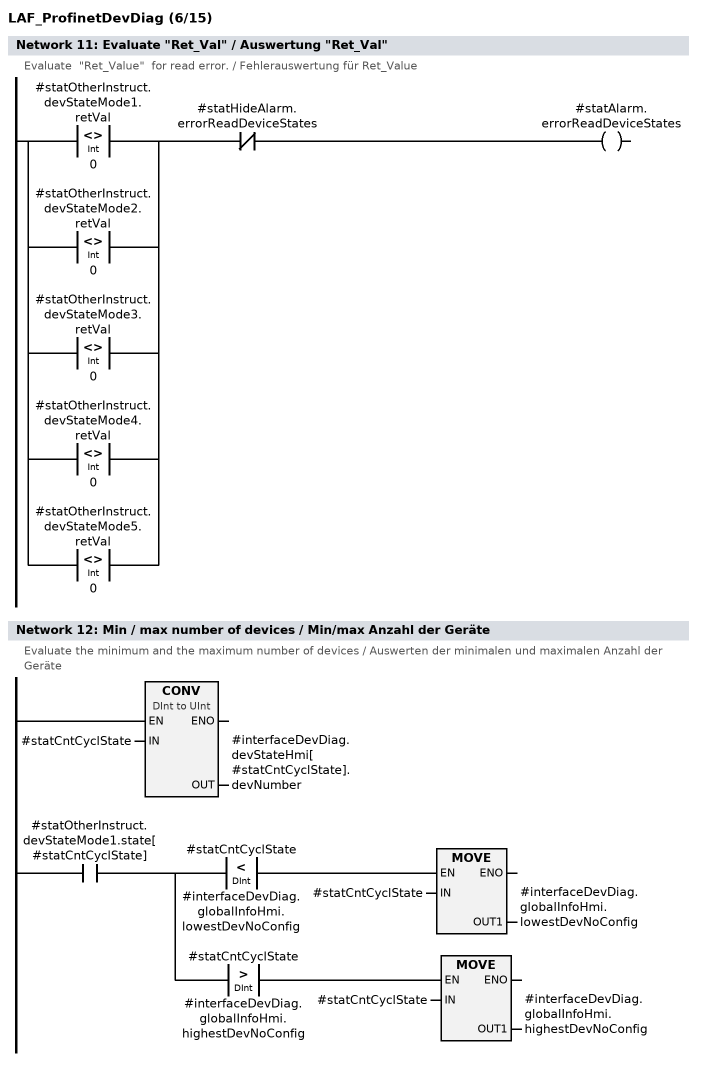
   RUNG wire#powerrail
      { S7_Templates := "SrcType := Int" } NE_Contact(in1 := #statOtherInstruct.devStateMode1.retVal, in2 := 0)
      wire#w1
      I_Contact( #statHideAlarm.errorReadDeviceStates )
      Coil( #statAlarm.errorReadDeviceStates )
   END_RUNG
   RUNG wire#powerrail
      { S7_Templates := "SrcType := Int" } NE_Contact(in1 := #statOtherInstruct.devStateMode2.retVal, in2 := 0)
   END_RUNG wire#w1
   RUNG wire#powerrail
      { S7_Templates := "SrcType := Int" } NE_Contact(in1 := #statOtherInstruct.devStateMode3.retVal, in2 := 0)
   END_RUNG wire#w1
   RUNG wire#powerrail
      { S7_Templates := "SrcType := Int" } NE_Contact(in1 := #statOtherInstruct.devStateMode4.retVal, in2 := 0)
   END_RUNG wire#w1
   RUNG wire#powerrail
      { S7_Templates := "SrcType := Int" } NE_Contact(in1 := #statOtherInstruct.devStateMode5.retVal, in2 := 0)
   END_RUNG wire#w1
   // the same network as SCL:
   #statAlarm.errorReadDeviceStates := ((#statOtherInstruct.devStateMode1.retVal <> 0) OR (#statOtherInstruct.devStateMode2.retVal <> 0) OR (#statOtherInstruct.devStateMode3.retVal <> 0) OR (#statOtherInstruct.devStateMode4.retVal <> 0) OR (#statOtherInstruct.devStateMode5.retVal <> 0)) AND NOT #statHideAlarm.errorReadDeviceStates;
END_REGION

REGION Network 12: Min / max number of devices / Min/max Anzahl der Geräte
   // Evaluate the minimum and the maximum number of devices / Auswerten der minimalen und maximalen Anzahl der Geräte
   RUNG wire#powerrail
      { S7_Templates := "[SrcType := DInt, DestType := UInt]" } Convert(in := #statCntCyclState, out => #interfaceDevDiag.devStateHmi[#statCntCyclState].devNumber)
   END_RUNG
   RUNG wire#powerrail
      Contact( #statOtherInstruct.devStateMode1.state[#statCntCyclState] )
      wire#w1
      { S7_Templates := "SrcType := DInt" } LT_Contact(in1 := #statCntCyclState, in2 := #interfaceDevDiag.globalInfoHmi.lowestDevNoConfig)
      Move(in := #statCntCyclState, out1 => #interfaceDevDiag.globalInfoHmi.lowestDevNoConfig)
   END_RUNG
   RUNG wire#w1
      { S7_Templates := "SrcType := DInt" } GT_Contact(in1 := #statCntCyclState, in2 := #interfaceDevDiag.globalInfoHmi.highestDevNoConfig)
      Move(in := #statCntCyclState, out1 => #interfaceDevDiag.globalInfoHmi.highestDevNoConfig)
   END_RUNG
   // the same network as SCL:
   #interfaceDevDiag.devStateHmi[#statCntCyclState].devNumber := DINT_TO_UINT(#statCntCyclState);
   IF #statOtherInstruct.devStateMode1.state[#statCntCyclState] AND (#statCntCyclState < #interfaceDevDiag.globalInfoHmi.lowestDevNoConfig) THEN
       #interfaceDevDiag.globalInfoHmi.lowestDevNoConfig := #statCntCyclState;
   END_IF;
   IF #statOtherInstruct.devStateMode1.state[#statCntCyclState] AND (#statCntCyclState > #interfaceDevDiag.globalInfoHmi.highestDevNoConfig) THEN
       #interfaceDevDiag.globalInfoHmi.highestDevNoConfig := #statCntCyclState;
   END_IF;
END_REGION

REGION Network 13: DeviceState 1..5
   // Evaluation and distribution of the deviceState 1..5 / DeviceStates_Mode2..5 auswerten und in Device-arrays schreiben
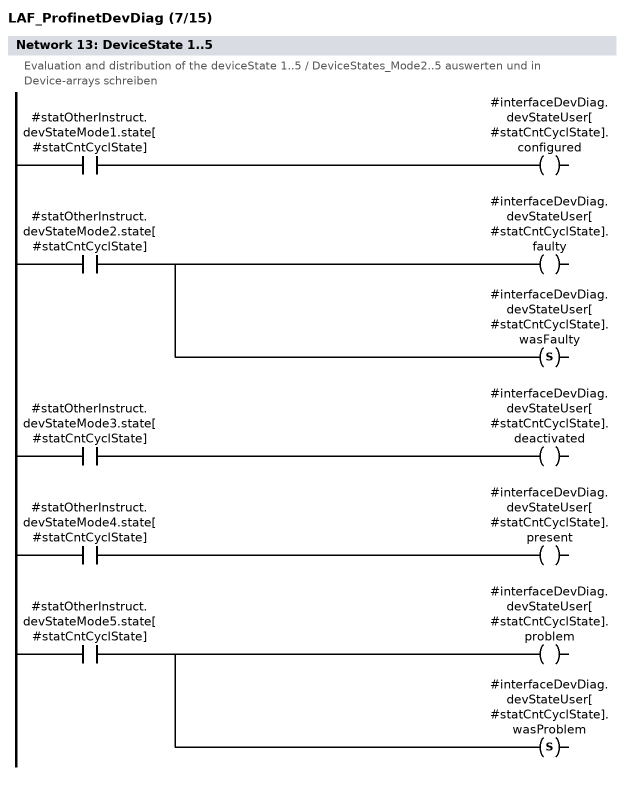
   RUNG wire#powerrail
      Contact( #statOtherInstruct.devStateMode1.state[#statCntCyclState] )
      Coil( #interfaceDevDiag.devStateUser[#statCntCyclState].configured )
   END_RUNG
   RUNG wire#powerrail
      Contact( #statOtherInstruct.devStateMode2.state[#statCntCyclState] )
      wire#w1
      Coil( #interfaceDevDiag.devStateUser[#statCntCyclState].faulty )
   END_RUNG
   RUNG wire#w1
      S_Coil( #interfaceDevDiag.devStateUser[#statCntCyclState].wasFaulty )
   END_RUNG
   RUNG wire#powerrail
      Contact( #statOtherInstruct.devStateMode3.state[#statCntCyclState] )
      Coil( #interfaceDevDiag.devStateUser[#statCntCyclState].deactivated )
   END_RUNG
   RUNG wire#powerrail
      Contact( #statOtherInstruct.devStateMode4.state[#statCntCyclState] )
      Coil( #interfaceDevDiag.devStateUser[#statCntCyclState].present )
   END_RUNG
   RUNG wire#powerrail
      Contact( #statOtherInstruct.devStateMode5.state[#statCntCyclState] )
      wire#w2
      Coil( #interfaceDevDiag.devStateUser[#statCntCyclState].problem )
   END_RUNG
   RUNG wire#w2
      S_Coil( #interfaceDevDiag.devStateUser[#statCntCyclState].wasProblem )
   END_RUNG
   // the same network as SCL:
   #interfaceDevDiag.devStateUser[#statCntCyclState].configured := #statOtherInstruct.devStateMode1.state[#statCntCyclState];
   #_w1 := #statOtherInstruct.devStateMode2.state[#statCntCyclState];
   #interfaceDevDiag.devStateUser[#statCntCyclState].faulty := #statOtherInstruct.devStateMode2.state[#statCntCyclState];
   IF #_w1 THEN #interfaceDevDiag.devStateUser[#statCntCyclState].wasFaulty := TRUE; END_IF;
   #interfaceDevDiag.devStateUser[#statCntCyclState].deactivated := #statOtherInstruct.devStateMode3.state[#statCntCyclState];
   #interfaceDevDiag.devStateUser[#statCntCyclState].present := #statOtherInstruct.devStateMode4.state[#statCntCyclState];
   #_w2 := #statOtherInstruct.devStateMode5.state[#statCntCyclState];
   #interfaceDevDiag.devStateUser[#statCntCyclState].problem := #statOtherInstruct.devStateMode5.state[#statCntCyclState];
   IF #_w2 THEN #interfaceDevDiag.devStateUser[#statCntCyclState].wasProblem := TRUE; END_IF;
END_REGION

REGION Network 14: DeviceState handover decimal coded and create counter / Device-Status: dez. codiert übergeben und Zähler bilden
   // State/Wert    Hintergrund     Vordergrund/Text// - Konfiguriert/Configrured//   und nicht Faulty//   und nicht Deaktivated//   und Present//   und nicht Problem//   und nicht WasFaulty//   und nicht WasProblem..................1........Grün............Schwarz// - Fehler/Faulty//   und Configured//   und Present....................................2........Rot.............Schwarz// - Deaktiviert/Deaktivated...............3........Weiß............Schwarz// - nicht Vorhanden/Present//   und Configured..............................4........Blau............Rot// - Problem/Problem//   und Configured//   und Present....................................5........Orange..........Schwarz// - WarGestört/WasFaulty..................6........Grün............Rot// - WarProblem/WasProblem............7........Grün............Orange//--------------------------------------------------//Dez. State: 1
   // State/Wert    Hintergrund     Vordergrund/Text
   // // - Konfiguriert/Configrured
   // //   und nicht Faulty
   // //   und nicht Deaktivated
   // //   und Present
   // //   und nicht Problem
   // //   und nicht WasFaulty
   // //   und nicht WasProblem..................1........Grün............Schwarz
   // // - Fehler/Faulty
   // //   und Configured
   // //   und Present....................................2........Rot.............Schwarz
   // // - Deaktiviert/Deaktivated...............3........Weiß............Schwarz
   // // - nicht Vorhanden/Present
   // //   und Configured..............................4........Blau............Rot
   // // - Problem/Problem
   // //   und Configured
   // //   und Present....................................5........Orange..........Schwarz
   // // - WarGestört/WasFaulty..................6........Grün............Rot
   // // - WarProblem/WasProblem............7........Grün............Orange
   // //--------------------------------------------------
   // //Dez. State: 1
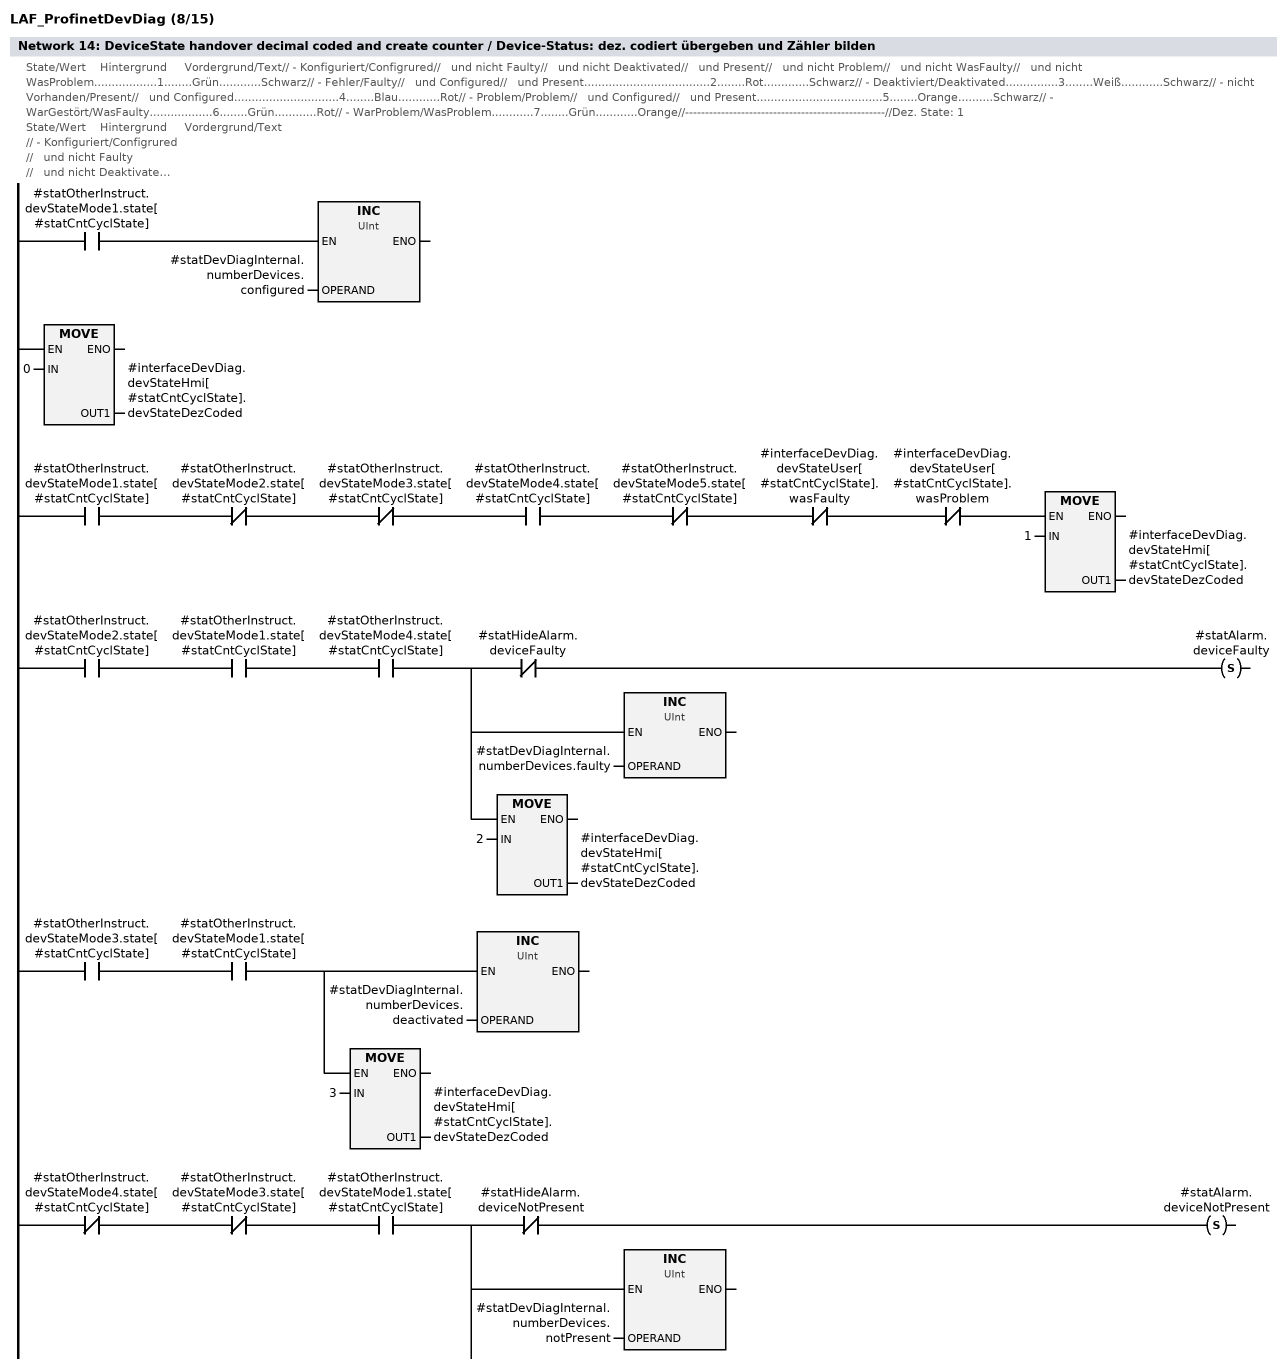
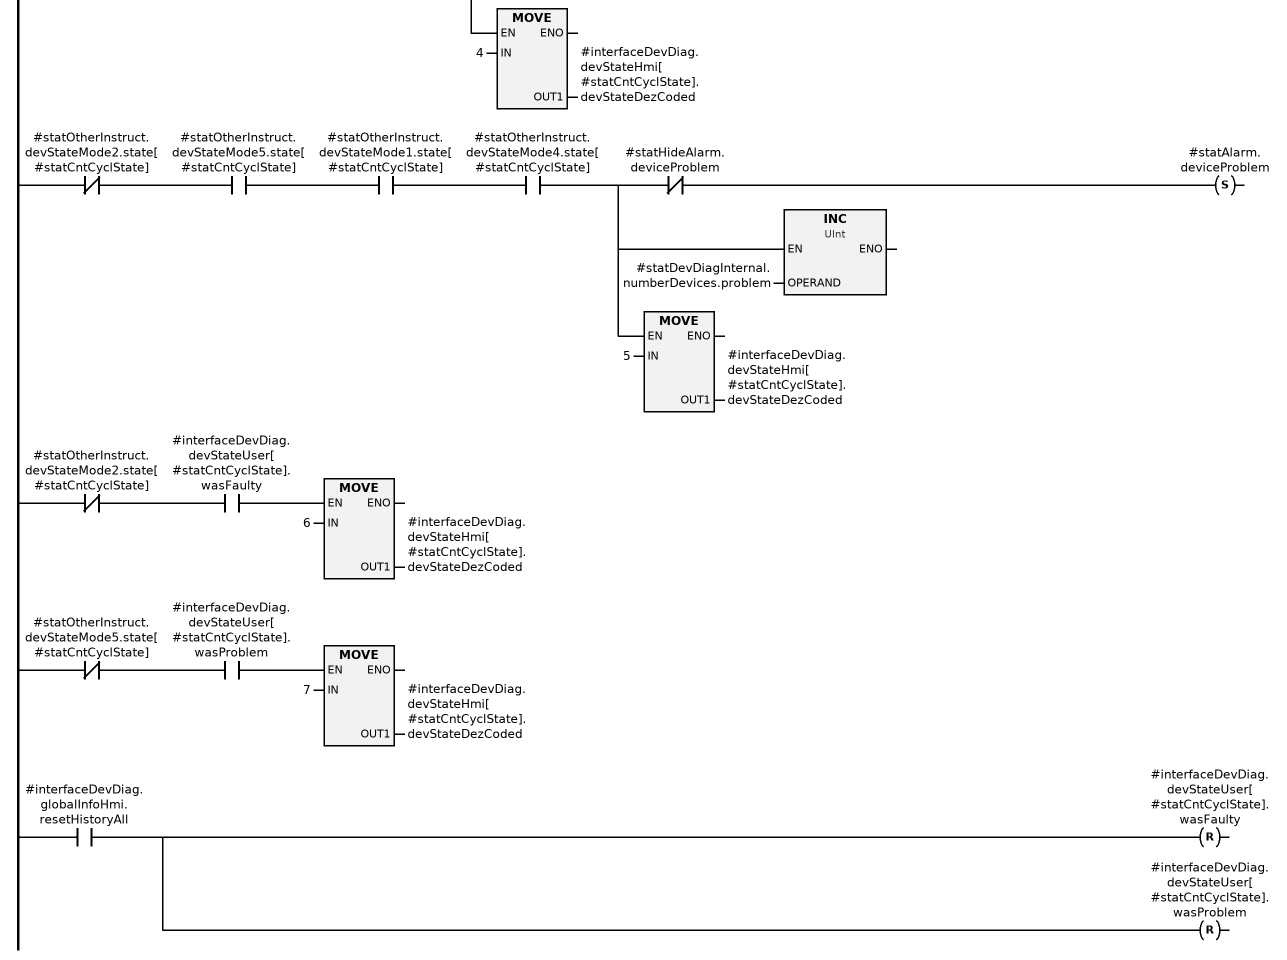
   RUNG wire#powerrail
      Contact( #statOtherInstruct.devStateMode1.state[#statCntCyclState] )
      { S7_Templates := "DestType := UInt" } Inc( #statDevDiagInternal.numberDevices.configured )
   END_RUNG
   RUNG wire#powerrail
      Move(in := 0, out1 => #interfaceDevDiag.devStateHmi[#statCntCyclState].devStateDezCoded)
   END_RUNG
   RUNG wire#powerrail
      Contact( #statOtherInstruct.devStateMode1.state[#statCntCyclState] )
      I_Contact( #statOtherInstruct.devStateMode2.state[#statCntCyclState] )
      I_Contact( #statOtherInstruct.devStateMode3.state[#statCntCyclState] )
      Contact( #statOtherInstruct.devStateMode4.state[#statCntCyclState] )
      I_Contact( #statOtherInstruct.devStateMode5.state[#statCntCyclState] )
      I_Contact( #interfaceDevDiag.devStateUser[#statCntCyclState].wasFaulty )
      I_Contact( #interfaceDevDiag.devStateUser[#statCntCyclState].wasProblem )
      Move(in := 1, out1 => #interfaceDevDiag.devStateHmi[#statCntCyclState].devStateDezCoded)
   END_RUNG
   RUNG wire#powerrail
      Contact( #statOtherInstruct.devStateMode2.state[#statCntCyclState] )
      Contact( #statOtherInstruct.devStateMode1.state[#statCntCyclState] )
      Contact( #statOtherInstruct.devStateMode4.state[#statCntCyclState] )
      wire#w1
      I_Contact( #statHideAlarm.deviceFaulty )
      S_Coil( #statAlarm.deviceFaulty )
   END_RUNG
   RUNG wire#w1
      { S7_Templates := "DestType := UInt" } Inc( #statDevDiagInternal.numberDevices.faulty )
   END_RUNG
   RUNG wire#w1
      Move(in := 2, out1 => #interfaceDevDiag.devStateHmi[#statCntCyclState].devStateDezCoded)
   END_RUNG
   RUNG wire#powerrail
      Contact( #statOtherInstruct.devStateMode3.state[#statCntCyclState] )
      Contact( #statOtherInstruct.devStateMode1.state[#statCntCyclState] )
      wire#w2
      { S7_Templates := "DestType := UInt" } Inc( #statDevDiagInternal.numberDevices.deactivated )
   END_RUNG
   RUNG wire#w2
      Move(in := 3, out1 => #interfaceDevDiag.devStateHmi[#statCntCyclState].devStateDezCoded)
   END_RUNG
   RUNG wire#powerrail
      I_Contact( #statOtherInstruct.devStateMode4.state[#statCntCyclState] )
      I_Contact( #statOtherInstruct.devStateMode3.state[#statCntCyclState] )
      Contact( #statOtherInstruct.devStateMode1.state[#statCntCyclState] )
      wire#w3
      I_Contact( #statHideAlarm.deviceNotPresent )
      S_Coil( #statAlarm.deviceNotPresent )
   END_RUNG
   RUNG wire#w3
      { S7_Templates := "DestType := UInt" } Inc( #statDevDiagInternal.numberDevices.notPresent )
   END_RUNG
   RUNG wire#w3
      Move(in := 4, out1 => #interfaceDevDiag.devStateHmi[#statCntCyclState].devStateDezCoded)
   END_RUNG
   RUNG wire#powerrail
      I_Contact( #statOtherInstruct.devStateMode2.state[#statCntCyclState] )
      Contact( #statOtherInstruct.devStateMode5.state[#statCntCyclState] )
      Contact( #statOtherInstruct.devStateMode1.state[#statCntCyclState] )
      Contact( #statOtherInstruct.devStateMode4.state[#statCntCyclState] )
      wire#w4
      I_Contact( #statHideAlarm.deviceProblem )
      S_Coil( #statAlarm.deviceProblem )
   END_RUNG
   RUNG wire#w4
      { S7_Templates := "DestType := UInt" } Inc( #statDevDiagInternal.numberDevices.problem )
   END_RUNG
   RUNG wire#w4
      Move(in := 5, out1 => #interfaceDevDiag.devStateHmi[#statCntCyclState].devStateDezCoded)
   END_RUNG
   RUNG wire#powerrail
      I_Contact( #statOtherInstruct.devStateMode2.state[#statCntCyclState] )
      Contact( #interfaceDevDiag.devStateUser[#statCntCyclState].wasFaulty )
      Move(in := 6, out1 => #interfaceDevDiag.devStateHmi[#statCntCyclState].devStateDezCoded)
   END_RUNG
   RUNG wire#powerrail
      I_Contact( #statOtherInstruct.devStateMode5.state[#statCntCyclState] )
      Contact( #interfaceDevDiag.devStateUser[#statCntCyclState].wasProblem )
      Move(in := 7, out1 => #interfaceDevDiag.devStateHmi[#statCntCyclState].devStateDezCoded)
   END_RUNG
   RUNG wire#powerrail
      Contact( #interfaceDevDiag.globalInfoHmi.resetHistoryAll )
      wire#w5
      R_Coil( #interfaceDevDiag.devStateUser[#statCntCyclState].wasFaulty )
   END_RUNG
   RUNG wire#w5
      R_Coil( #interfaceDevDiag.devStateUser[#statCntCyclState].wasProblem )
   END_RUNG
   // the same network as SCL:
   IF #statOtherInstruct.devStateMode1.state[#statCntCyclState] THEN
       #statDevDiagInternal.numberDevices.configured := #statDevDiagInternal.numberDevices.configured + 1;
   END_IF;
   #interfaceDevDiag.devStateHmi[#statCntCyclState].devStateDezCoded := 0;
   IF #statOtherInstruct.devStateMode1.state[#statCntCyclState] AND NOT #statOtherInstruct.devStateMode2.state[#statCntCyclState] AND NOT #statOtherInstruct.devStateMode3.state[#statCntCyclState] AND #statOtherInstruct.devStateMode4.state[#statCntCyclState] AND NOT #statOtherInstruct.devStateMode5.state[#statCntCyclState] AND NOT #interfaceDevDiag.devStateUser[#statCntCyclState].wasFaulty AND NOT #interfaceDevDiag.devStateUser[#statCntCyclState].wasProblem THEN
       #interfaceDevDiag.devStateHmi[#statCntCyclState].devStateDezCoded := 1;
   END_IF;
   #_w1 := #statOtherInstruct.devStateMode2.state[#statCntCyclState] AND #statOtherInstruct.devStateMode1.state[#statCntCyclState] AND #statOtherInstruct.devStateMode4.state[#statCntCyclState];
   IF #_w1 AND NOT #statHideAlarm.deviceFaulty THEN #statAlarm.deviceFaulty := TRUE; END_IF;
   IF #_w1 THEN
       #statDevDiagInternal.numberDevices.faulty := #statDevDiagInternal.numberDevices.faulty + 1;
       #interfaceDevDiag.devStateHmi[#statCntCyclState].devStateDezCoded := 2;
   END_IF;
   IF #statOtherInstruct.devStateMode3.state[#statCntCyclState] AND #statOtherInstruct.devStateMode1.state[#statCntCyclState] THEN
       #statDevDiagInternal.numberDevices.deactivated := #statDevDiagInternal.numberDevices.deactivated + 1;
       #interfaceDevDiag.devStateHmi[#statCntCyclState].devStateDezCoded := 3;
   END_IF;
   #_w2 := NOT #statOtherInstruct.devStateMode4.state[#statCntCyclState] AND NOT #statOtherInstruct.devStateMode3.state[#statCntCyclState] AND #statOtherInstruct.devStateMode1.state[#statCntCyclState];
   IF #_w2 AND NOT #statHideAlarm.deviceNotPresent THEN #statAlarm.deviceNotPresent := TRUE; END_IF;
   IF #_w2 THEN
       #statDevDiagInternal.numberDevices.notPresent := #statDevDiagInternal.numberDevices.notPresent + 1;
       #interfaceDevDiag.devStateHmi[#statCntCyclState].devStateDezCoded := 4;
   END_IF;
   #_w3 := NOT #statOtherInstruct.devStateMode2.state[#statCntCyclState] AND #statOtherInstruct.devStateMode5.state[#statCntCyclState] AND #statOtherInstruct.devStateMode1.state[#statCntCyclState] AND #statOtherInstruct.devStateMode4.state[#statCntCyclState];
   IF #_w3 AND NOT #statHideAlarm.deviceProblem THEN #statAlarm.deviceProblem := TRUE; END_IF;
   IF #_w3 THEN
       #statDevDiagInternal.numberDevices.problem := #statDevDiagInternal.numberDevices.problem + 1;
       #interfaceDevDiag.devStateHmi[#statCntCyclState].devStateDezCoded := 5;
   END_IF;
   IF NOT #statOtherInstruct.devStateMode2.state[#statCntCyclState] AND #interfaceDevDiag.devStateUser[#statCntCyclState].wasFaulty THEN
       #interfaceDevDiag.devStateHmi[#statCntCyclState].devStateDezCoded := 6;
   END_IF;
   IF NOT #statOtherInstruct.devStateMode5.state[#statCntCyclState] AND #interfaceDevDiag.devStateUser[#statCntCyclState].wasProblem THEN
       #interfaceDevDiag.devStateHmi[#statCntCyclState].devStateDezCoded := 7;
   END_IF;
   IF #interfaceDevDiag.globalInfoHmi.resetHistoryAll THEN
       #interfaceDevDiag.devStateUser[#statCntCyclState].wasFaulty := FALSE;
       #interfaceDevDiag.devStateUser[#statCntCyclState].wasProblem := FALSE;
   END_IF;
END_REGION

REGION Network 15: Reset error counter / Rücksetzen des Fehlerzählers
   // Reset DeviceErrorCounter and resetHistoryAll from HMI / Rücksetzten des DeviceErrorCounter und resetHistoryAll vom HMI
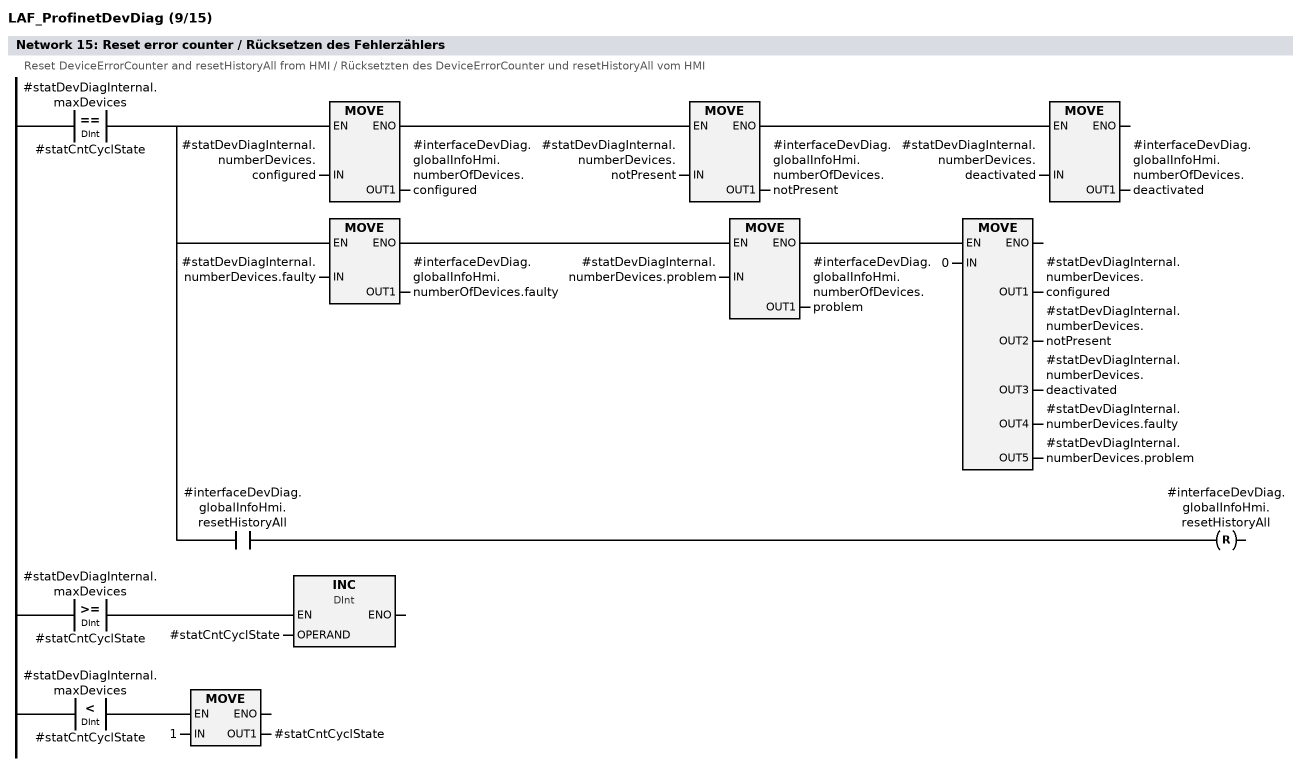
   RUNG wire#powerrail
      { S7_Templates := "SrcType := DInt" } EQ_Contact(in1 := #statDevDiagInternal.maxDevices, in2 := #statCntCyclState)
      wire#w1
      Move(in := #statDevDiagInternal.numberDevices.configured, out1 => #interfaceDevDiag.globalInfoHmi.numberOfDevices.configured)
      Move(in := #statDevDiagInternal.numberDevices.notPresent, out1 => #interfaceDevDiag.globalInfoHmi.numberOfDevices.notPresent)
      Move(in := #statDevDiagInternal.numberDevices.deactivated, out1 => #interfaceDevDiag.globalInfoHmi.numberOfDevices.deactivated)
   END_RUNG
   RUNG wire#w1
      Move(in := #statDevDiagInternal.numberDevices.faulty, out1 => #interfaceDevDiag.globalInfoHmi.numberOfDevices.faulty)
      Move(in := #statDevDiagInternal.numberDevices.problem, out1 => #interfaceDevDiag.globalInfoHmi.numberOfDevices.problem)
      Move(in := 0, out1 => #statDevDiagInternal.numberDevices.configured, out2 => #statDevDiagInternal.numberDevices.notPresent, out3 => #statDevDiagInternal.numberDevices.deactivated, out4 => #statDevDiagInternal.numberDevices.faulty, out5 => #statDevDiagInternal.numberDevices.problem)
   END_RUNG
   RUNG wire#w1
      Contact( #interfaceDevDiag.globalInfoHmi.resetHistoryAll )
      R_Coil( #interfaceDevDiag.globalInfoHmi.resetHistoryAll )
   END_RUNG
   RUNG wire#powerrail
      { S7_Templates := "SrcType := DInt" } GE_Contact(in1 := #statDevDiagInternal.maxDevices, in2 := #statCntCyclState)
      { S7_Templates := "DestType := DInt" } Inc( #statCntCyclState )
   END_RUNG
   RUNG wire#powerrail
      { S7_Templates := "SrcType := DInt" } LT_Contact(in1 := #statDevDiagInternal.maxDevices, in2 := #statCntCyclState)
      Move(in := 1, out1 => #statCntCyclState)
   END_RUNG
   // the same network as SCL:
   #_w1 := #statDevDiagInternal.maxDevices = #statCntCyclState;
   IF #_w1 THEN
       #interfaceDevDiag.globalInfoHmi.numberOfDevices.configured := #statDevDiagInternal.numberDevices.configured;
       #interfaceDevDiag.globalInfoHmi.numberOfDevices.notPresent := #statDevDiagInternal.numberDevices.notPresent;
       #interfaceDevDiag.globalInfoHmi.numberOfDevices.deactivated := #statDevDiagInternal.numberDevices.deactivated;
       #interfaceDevDiag.globalInfoHmi.numberOfDevices.faulty := #statDevDiagInternal.numberDevices.faulty;
       #interfaceDevDiag.globalInfoHmi.numberOfDevices.problem := #statDevDiagInternal.numberDevices.problem;
       #statDevDiagInternal.numberDevices.configured := 0;
       #statDevDiagInternal.numberDevices.notPresent := 0;
       #statDevDiagInternal.numberDevices.deactivated := 0;
       #statDevDiagInternal.numberDevices.faulty := 0;
       #statDevDiagInternal.numberDevices.problem := 0;
   END_IF;
   IF #_w1 AND #interfaceDevDiag.globalInfoHmi.resetHistoryAll THEN
       #interfaceDevDiag.globalInfoHmi.resetHistoryAll := FALSE;
   END_IF;
   IF #statDevDiagInternal.maxDevices >= #statCntCyclState THEN
       #statCntCyclState := #statCntCyclState + 1;
   END_IF;
   IF #statDevDiagInternal.maxDevices < #statCntCyclState THEN #statCntCyclState := 1; END_IF;
END_REGION

REGION Network 16: Read device name / Lesen des Gerätenamens
   // Once only read of device names "Get_Name" / Einmaliges Lesen: Get_Name: Name des Devices lesen
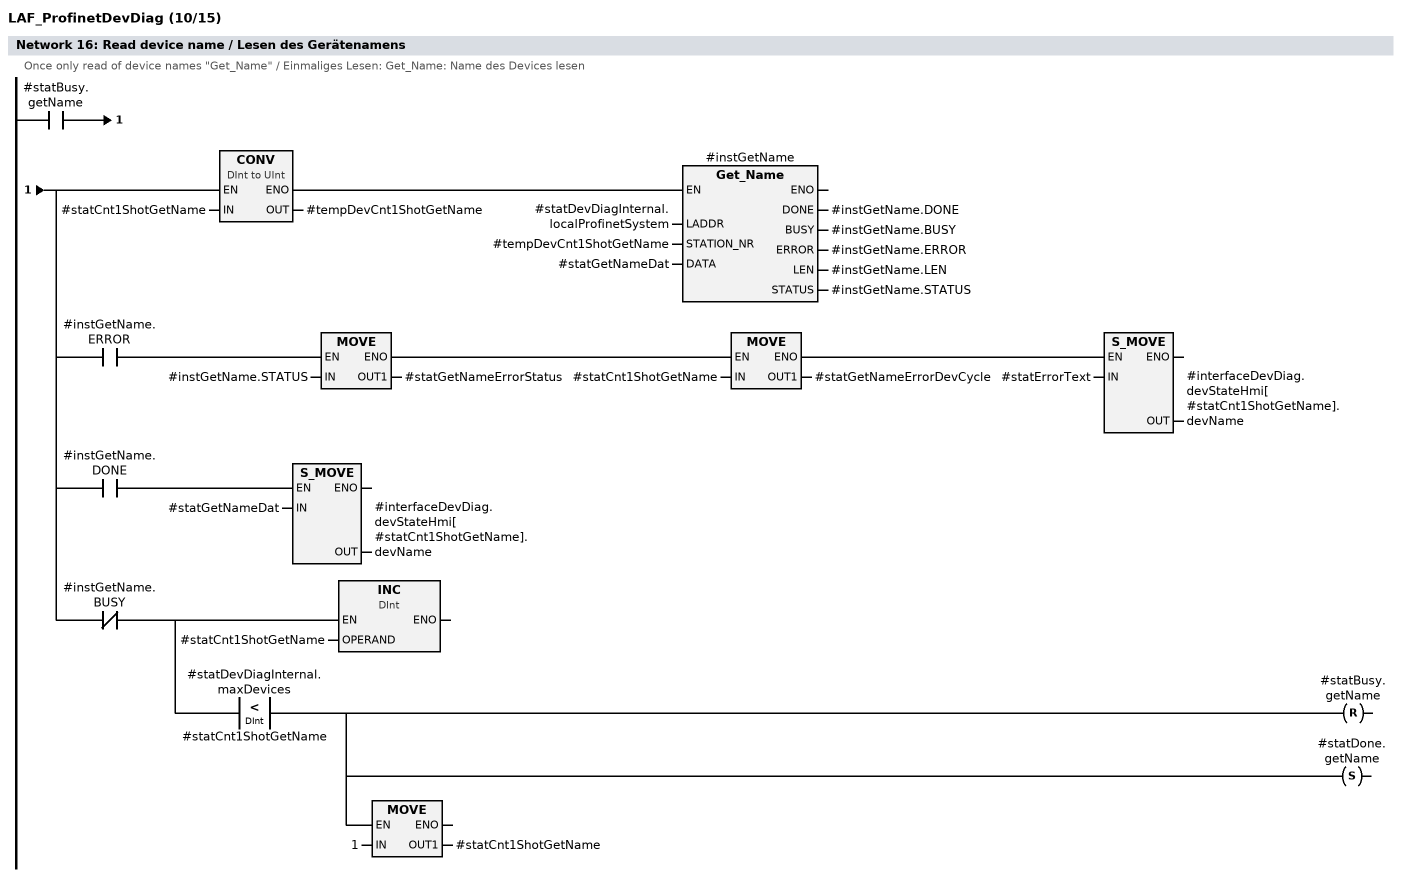
   RUNG wire#powerrail
      Contact( #statBusy.getName )
      wire#w1
      { S7_Templates := "[SrcType := DInt, DestType := UInt]" } Convert(in := #statCnt1ShotGetName, out => #tempDevCnt1ShotGetName)
      #instGetName.Get_Name(LADDR := #statDevDiagInternal.localProfinetSystem, STATION_NR := #tempDevCnt1ShotGetName, DATA := #statGetNameDat, DONE => #instGetName.DONE, BUSY => #instGetName.BUSY, ERROR => #instGetName.ERROR, LEN => #instGetName.LEN, STATUS => #instGetName.STATUS)
   END_RUNG
   RUNG wire#w1
      Contact( #instGetName.ERROR )
      Move(in := #instGetName.STATUS, out1 => #statGetNameErrorStatus)
      Move(in := #statCnt1ShotGetName, out1 => #statGetNameErrorDevCycle)
      S_Move(in := #statErrorText, out => #interfaceDevDiag.devStateHmi[#statCnt1ShotGetName].devName)
   END_RUNG
   RUNG wire#w1
      Contact( #instGetName.DONE )
      S_Move(in := #statGetNameDat, out => #interfaceDevDiag.devStateHmi[#statCnt1ShotGetName].devName)
   END_RUNG
   RUNG wire#w1
      I_Contact( #instGetName.BUSY )
      wire#w2
      { S7_Templates := "DestType := DInt" } Inc( #statCnt1ShotGetName )
   END_RUNG
   RUNG wire#w2
      { S7_Templates := "SrcType := DInt" } LT_Contact(in1 := #statDevDiagInternal.maxDevices, in2 := #statCnt1ShotGetName)
      wire#w3
      R_Coil( #statBusy.getName )
   END_RUNG
   RUNG wire#w3
      S_Coil( #statDone.getName )
   END_RUNG
   RUNG wire#w3
      Move(in := 1, out1 => #statCnt1ShotGetName)
   END_RUNG
   // the same network as SCL:
   IF #statBusy.getName THEN
       #tempDevCnt1ShotGetName := DINT_TO_UINT(#statCnt1ShotGetName);
       #instGetName(LADDR := #statDevDiagInternal.localProfinetSystem,   // Get_Name
                    STATION_NR := #tempDevCnt1ShotGetName,
                    DATA := #statGetNameDat,
                    DONE => #instGetName.DONE,
                    BUSY => #instGetName.BUSY,
                    ERROR => #instGetName.ERROR,
                    LEN => #instGetName.LEN,
                    STATUS => #instGetName.STATUS);
   END_IF;
   IF #statBusy.getName AND #instGetName.ERROR THEN
       #statGetNameErrorStatus := #instGetName.STATUS;
       #statGetNameErrorDevCycle := #statCnt1ShotGetName;
       #interfaceDevDiag.devStateHmi[#statCnt1ShotGetName].devName := #statErrorText;
   END_IF;
   IF #statBusy.getName AND #instGetName.DONE THEN
       #interfaceDevDiag.devStateHmi[#statCnt1ShotGetName].devName := #statGetNameDat;
   END_IF;
   #_w1 := #statBusy.getName AND NOT #instGetName.BUSY;
   IF #_w1 THEN #statCnt1ShotGetName := #statCnt1ShotGetName + 1; END_IF;
   IF #_w1 AND (#statDevDiagInternal.maxDevices < #statCnt1ShotGetName) THEN
       #statBusy.getName := FALSE;
       #statDone.getName := TRUE;
       #statCnt1ShotGetName := 1;
   END_IF;
END_REGION

REGION Network 17: Once only read of "GEO2LOG" / Einmaliges Lesen: GEO2LOG: HW-Kennung des Devices ermitteln
   // HWTYPE=2 -> IO_Device, HWTYPE=5 -> Submodul
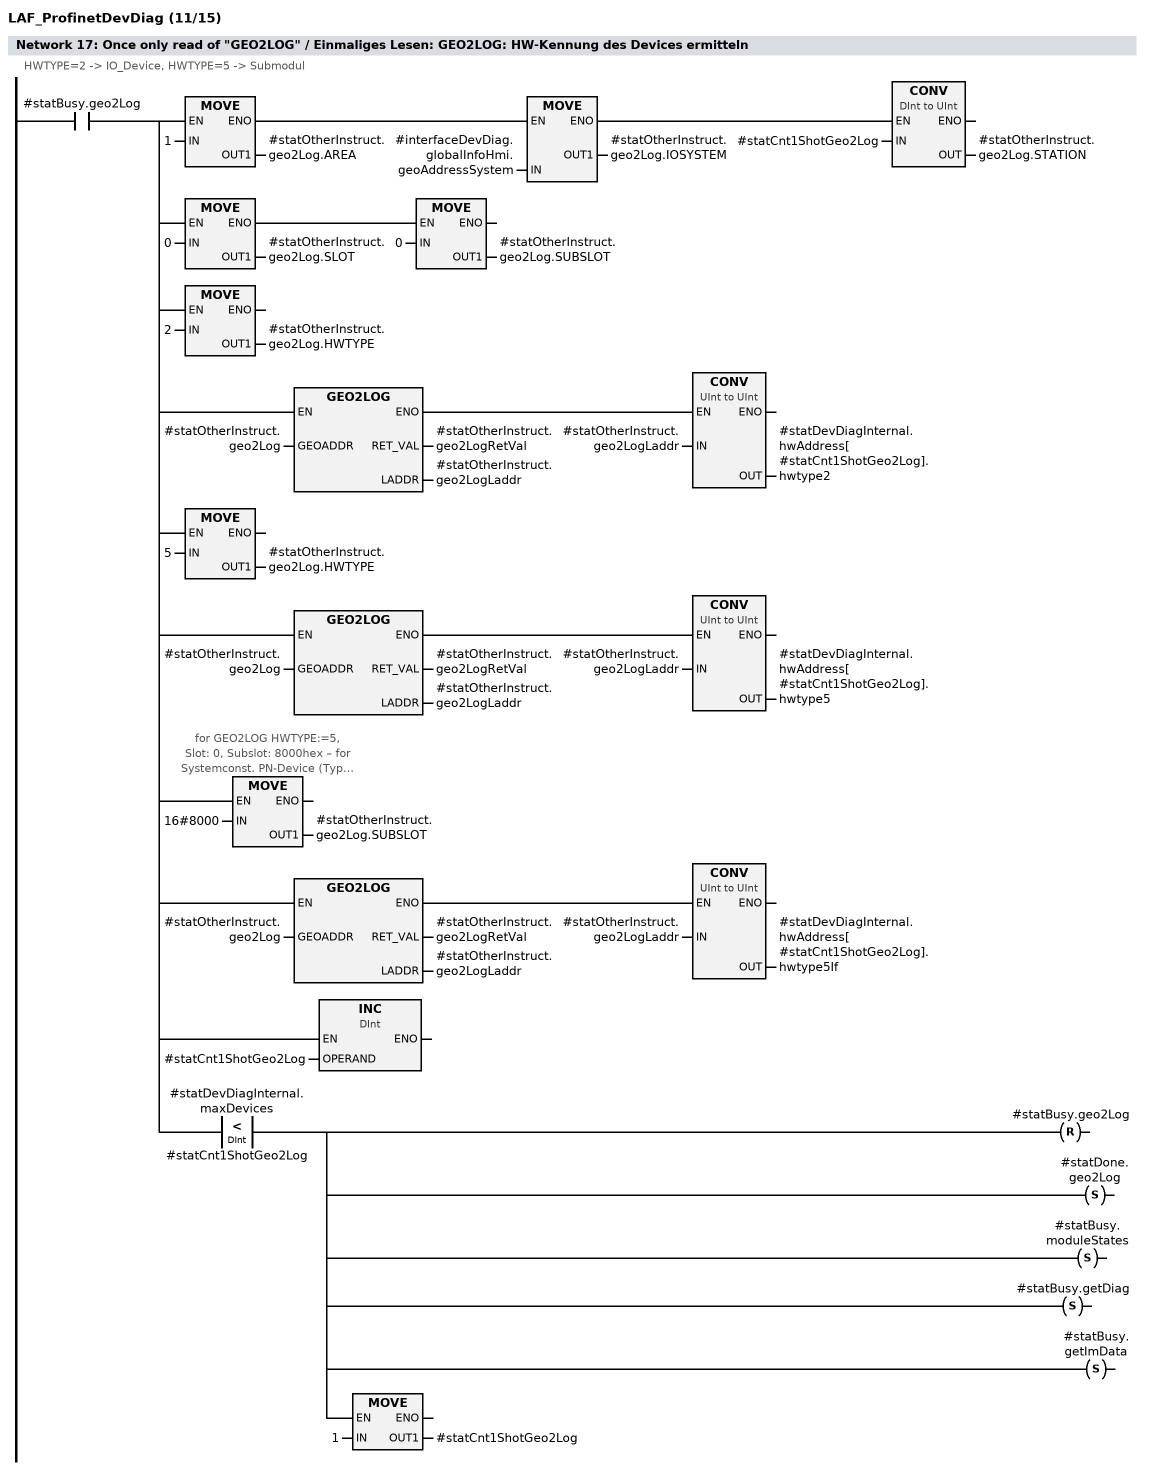
   RUNG wire#powerrail
      Contact( #statBusy.geo2Log )
      wire#w1
      Move(in := 1, out1 => #statOtherInstruct.geo2Log.AREA)
      Move(in := #interfaceDevDiag.globalInfoHmi.geoAddressSystem, out1 => #statOtherInstruct.geo2Log.IOSYSTEM)
      { S7_Templates := "[SrcType := DInt, DestType := UInt]" } Convert(in := #statCnt1ShotGeo2Log, out => #statOtherInstruct.geo2Log.STATION)
   END_RUNG
   RUNG wire#w1
      Move(in := 0, out1 => #statOtherInstruct.geo2Log.SLOT)
      Move(in := 0, out1 => #statOtherInstruct.geo2Log.SUBSLOT)
   END_RUNG
   RUNG wire#w1
      Move(in := 2, out1 => #statOtherInstruct.geo2Log.HWTYPE)
   END_RUNG
   RUNG wire#w1
      GEO2LOG(GEOADDR := #statOtherInstruct.geo2Log, RET_VAL => #statOtherInstruct.geo2LogRetVal, LADDR => #statOtherInstruct.geo2LogLaddr)
      { S7_Templates := "[SrcType := UInt, DestType := UInt]" } Convert(in := #statOtherInstruct.geo2LogLaddr, out => #statDevDiagInternal.hwAddress[#statCnt1ShotGeo2Log].hwtype2)
   END_RUNG
   RUNG wire#w1
      Move(in := 5, out1 => #statOtherInstruct.geo2Log.HWTYPE)
   END_RUNG
   RUNG wire#w1
      GEO2LOG(GEOADDR := #statOtherInstruct.geo2Log, RET_VAL => #statOtherInstruct.geo2LogRetVal, LADDR => #statOtherInstruct.geo2LogLaddr)
      { S7_Templates := "[SrcType := UInt, DestType := UInt]" } Convert(in := #statOtherInstruct.geo2LogLaddr, out => #statDevDiagInternal.hwAddress[#statCnt1ShotGeo2Log].hwtype5)
   END_RUNG
   RUNG wire#w1
      Move(in := 16#8000, out1 => #statOtherInstruct.geo2Log.SUBSLOT)   // for GEO2LOG HWTYPE:=5, Slot: 0, Subslot: 8000hex – for Systemconst. PN-Device (Typ: Hw_Interface) "...PROFINET-Schnittstelle" für GEO2LOG HWTYPE:=5, Slot: 0, Subslot: 8000hex – für Systemkonst. PN-Device (Typ: Hw_Interface) "...PROFINET-Schnittstelle"
   END_RUNG
   RUNG wire#w1
      GEO2LOG(GEOADDR := #statOtherInstruct.geo2Log, RET_VAL => #statOtherInstruct.geo2LogRetVal, LADDR => #statOtherInstruct.geo2LogLaddr)
      { S7_Templates := "[SrcType := UInt, DestType := UInt]" } Convert(in := #statOtherInstruct.geo2LogLaddr, out => #statDevDiagInternal.hwAddress[#statCnt1ShotGeo2Log].hwtype5If)
   END_RUNG
   RUNG wire#w1
      { S7_Templates := "DestType := DInt" } Inc( #statCnt1ShotGeo2Log )
   END_RUNG
   RUNG wire#w1
      { S7_Templates := "SrcType := DInt" } LT_Contact(in1 := #statDevDiagInternal.maxDevices, in2 := #statCnt1ShotGeo2Log)
      wire#w2
      R_Coil( #statBusy.geo2Log )
   END_RUNG
   RUNG wire#w2
      S_Coil( #statDone.geo2Log )
   END_RUNG
   RUNG wire#w2
      S_Coil( #statBusy.moduleStates )
   END_RUNG
   RUNG wire#w2
      S_Coil( #statBusy.getDiag )
   END_RUNG
   RUNG wire#w2
      S_Coil( #statBusy.getImData )
   END_RUNG
   RUNG wire#w2
      Move(in := 1, out1 => #statCnt1ShotGeo2Log)
   END_RUNG
   // the same network as SCL:
   IF #statBusy.geo2Log THEN
       #statOtherInstruct.geo2Log.AREA := 1;
       #statOtherInstruct.geo2Log.IOSYSTEM := #interfaceDevDiag.globalInfoHmi.geoAddressSystem;
       #statOtherInstruct.geo2Log.STATION := DINT_TO_UINT(#statCnt1ShotGeo2Log);
       #statOtherInstruct.geo2Log.SLOT := 0;
       #statOtherInstruct.geo2Log.SUBSLOT := 0;
       #statOtherInstruct.geo2Log.HWTYPE := 2;
   END_IF;
   #statOtherInstruct.geo2LogRetVal := GEO2LOG(EN := #statBusy.geo2Log,
                           GEOADDR := #statOtherInstruct.geo2Log,
                           LADDR => #statOtherInstruct.geo2LogLaddr,
                           ENO => #_w1);
   IF #_w1 THEN
       #statDevDiagInternal.hwAddress[#statCnt1ShotGeo2Log].hwtype2 := UINT_TO_UINT(#statOtherInstruct.geo2LogLaddr);
   END_IF;
   IF #statBusy.geo2Log THEN #statOtherInstruct.geo2Log.HWTYPE := 5; END_IF;
   #statOtherInstruct.geo2LogRetVal := GEO2LOG(EN := #statBusy.geo2Log,
                           GEOADDR := #statOtherInstruct.geo2Log,
                           LADDR => #statOtherInstruct.geo2LogLaddr,
                           ENO => #_w2);
   IF #_w2 THEN
       #statDevDiagInternal.hwAddress[#statCnt1ShotGeo2Log].hwtype5 := UINT_TO_UINT(#statOtherInstruct.geo2LogLaddr);
   END_IF;
   IF #statBusy.geo2Log THEN
       #statOtherInstruct.geo2Log.SUBSLOT := 16#8000;   // for GEO2LOG HWTYPE:=5, Slot: 0, Subslot: 8000hex – for Systemconst. PN-Device (Typ: Hw_Interface) "...PROFINET-Schnittstelle" für GEO2LOG HWTYPE:=5, Slot: 0, Subslot: 8000hex – für Systemkonst. PN-Device (Typ: Hw_Interface) "...PROFINET-Schnittstelle"
   END_IF;
   #statOtherInstruct.geo2LogRetVal := GEO2LOG(EN := #statBusy.geo2Log,
                           GEOADDR := #statOtherInstruct.geo2Log,
                           LADDR => #statOtherInstruct.geo2LogLaddr,
                           ENO => #_w3);
   IF #_w3 THEN
       #statDevDiagInternal.hwAddress[#statCnt1ShotGeo2Log].hwtype5If := UINT_TO_UINT(#statOtherInstruct.geo2LogLaddr);
   END_IF;
   IF #statBusy.geo2Log THEN #statCnt1ShotGeo2Log := #statCnt1ShotGeo2Log + 1; END_IF;
   #_w4 := #statBusy.geo2Log AND (#statDevDiagInternal.maxDevices < #statCnt1ShotGeo2Log);
   IF #_w4 THEN
       #statBusy.geo2Log := FALSE;
       #statDone.geo2Log := TRUE;
       #statBusy.moduleStates := TRUE;
       #statBusy.getDiag := TRUE;
       #statBusy.getImData := TRUE;
       #statCnt1ShotGeo2Log := 1;
   END_IF;
END_REGION

REGION Network 18: Read "ModulStates" / ModuleStates: Summenstatus/Modulfehler aller unterlagerten Module - mittels "ModuleStates" (Bit0)
   // Mode 2: faulty, Mode 5: problem, / Mode 2: gestoert, Mode 5: Problem,
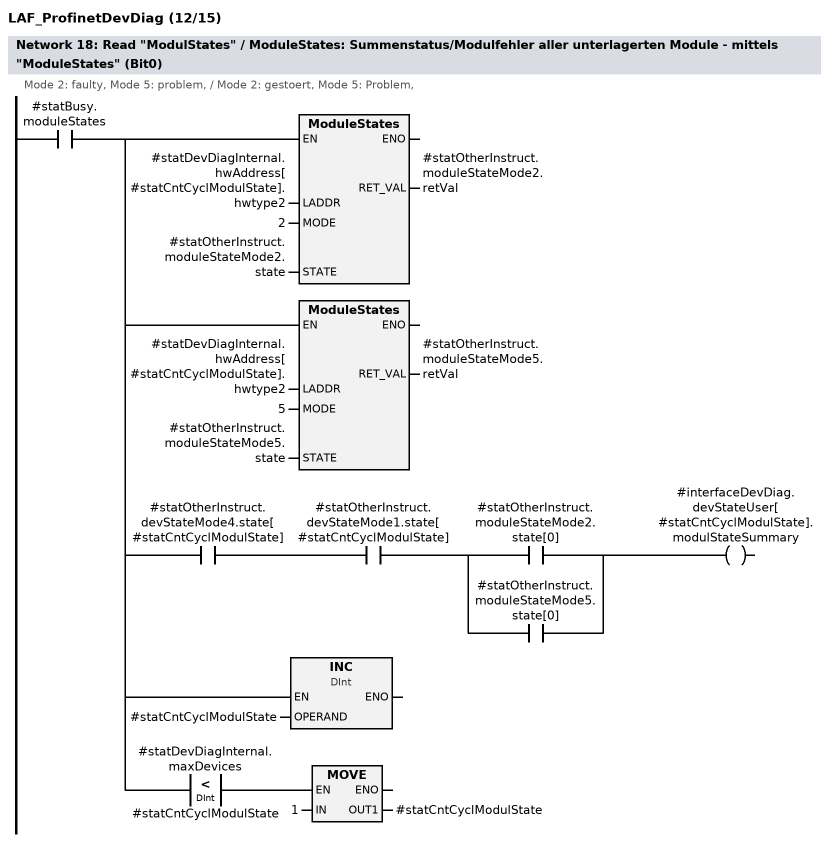
   RUNG wire#powerrail
      Contact( #statBusy.moduleStates )
      wire#w1
      ModuleStates(LADDR := #statDevDiagInternal.hwAddress[#statCntCyclModulState].hwtype2, MODE := 2, STATE := #statOtherInstruct.moduleStateMode2.state, Ret_Val => #statOtherInstruct.moduleStateMode2.retVal)
   END_RUNG
   RUNG wire#w1
      ModuleStates(LADDR := #statDevDiagInternal.hwAddress[#statCntCyclModulState].hwtype2, MODE := 5, STATE := #statOtherInstruct.moduleStateMode5.state, Ret_Val => #statOtherInstruct.moduleStateMode5.retVal)
   END_RUNG
   RUNG wire#w1
      Contact( #statOtherInstruct.devStateMode4.state[#statCntCyclModulState] )
      Contact( #statOtherInstruct.devStateMode1.state[#statCntCyclModulState] )
      wire#w2
      Contact( #statOtherInstruct.moduleStateMode2.state[0] )
      wire#w3
      Coil( #interfaceDevDiag.devStateUser[#statCntCyclModulState].modulStateSummary )
   END_RUNG
   RUNG wire#w2
      Contact( #statOtherInstruct.moduleStateMode5.state[0] )
   END_RUNG wire#w3
   RUNG wire#w1
      { S7_Templates := "DestType := DInt" } Inc( #statCntCyclModulState )
   END_RUNG
   RUNG wire#w1
      { S7_Templates := "SrcType := DInt" } LT_Contact(in1 := #statDevDiagInternal.maxDevices, in2 := #statCntCyclModulState)
      Move(in := 1, out1 => #statCntCyclModulState)
   END_RUNG
   // the same network as SCL:
   IF #statBusy.moduleStates THEN
       #statOtherInstruct.moduleStateMode2.retVal := ModuleStates(LADDR := #statDevDiagInternal.hwAddress[#statCntCyclModulState].hwtype2,
                               MODE := 2,
                               STATE := #statOtherInstruct.moduleStateMode2.state);
       #statOtherInstruct.moduleStateMode5.retVal := ModuleStates(LADDR := #statDevDiagInternal.hwAddress[#statCntCyclModulState].hwtype2,
                               MODE := 5,
                               STATE := #statOtherInstruct.moduleStateMode5.state);
   END_IF;
   #interfaceDevDiag.devStateUser[#statCntCyclModulState].modulStateSummary := #statBusy.moduleStates AND #statOtherInstruct.devStateMode4.state[#statCntCyclModulState] AND #statOtherInstruct.devStateMode1.state[#statCntCyclModulState] AND (#statOtherInstruct.moduleStateMode2.state[0] OR #statOtherInstruct.moduleStateMode5.state[0]);
   IF #statBusy.moduleStates THEN #statCntCyclModulState := #statCntCyclModulState + 1; END_IF;
   IF #statBusy.moduleStates AND (#statDevDiagInternal.maxDevices < #statCntCyclModulState) THEN
       #statCntCyclModulState := 1;
   END_IF;
END_REGION

REGION Network 19: GET_DIAG: Read Diagnostc informationen of a Hardware-Component / GET_DIAG: Diagnoseinformationen einer Hardware-Komponente auslesen
   // Mode 1
   // Mode1 ??? --- Mode2 noch testen, wenn nicht notwendig dann entfernen --- ???
   // #PNDeviceData.Internal.DevHWAddr_HWTYPE5_PNIF[#DEVCount_GET_DIAG_Cyclic]
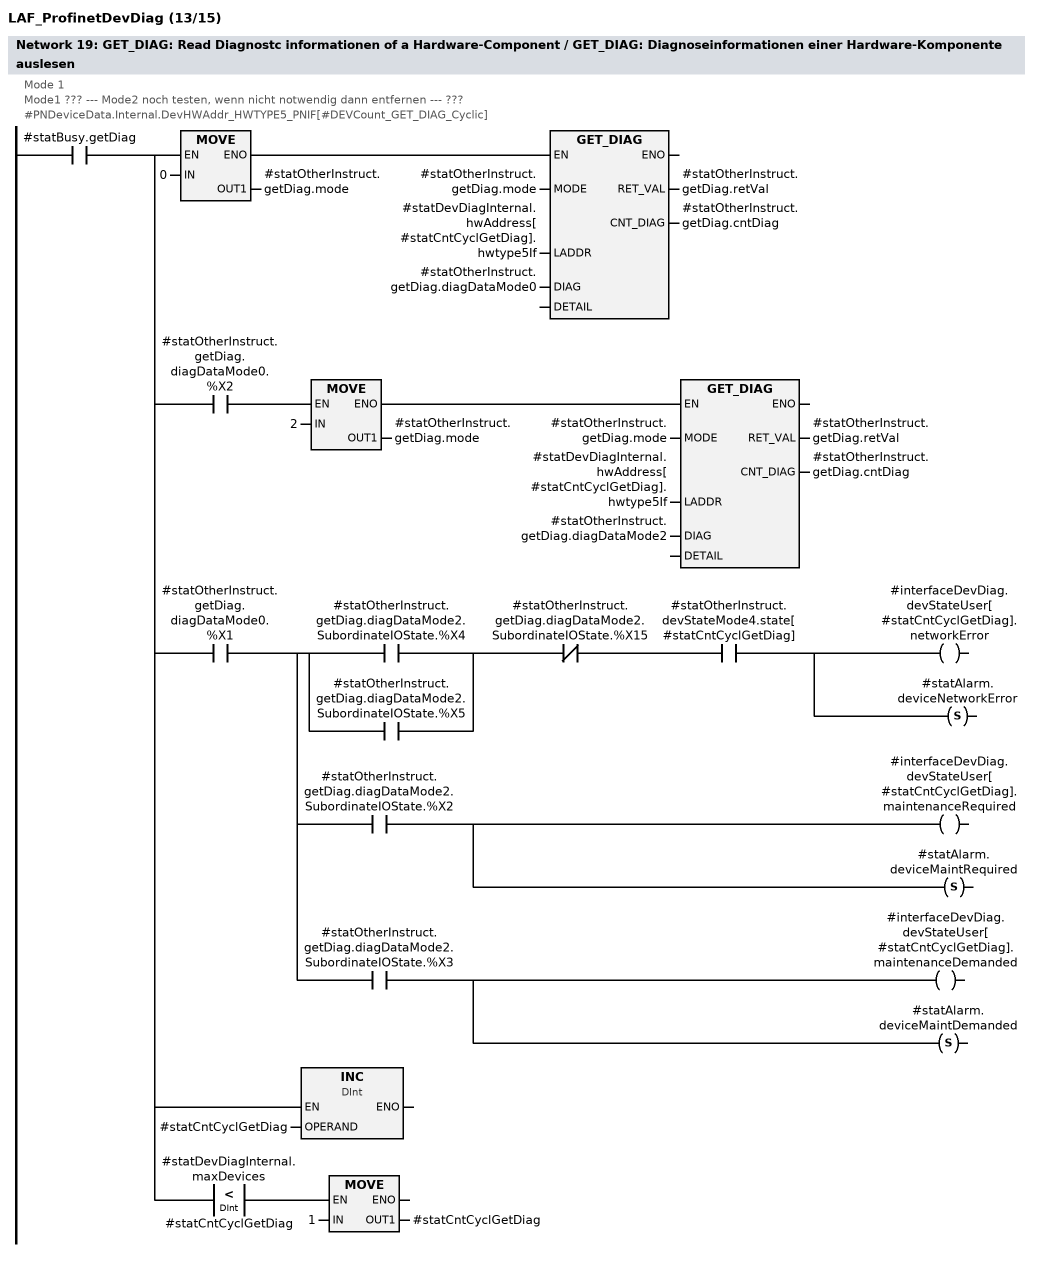
   RUNG wire#powerrail
      Contact( #statBusy.getDiag )
      wire#w1
      Move(in := 0, out1 => #statOtherInstruct.getDiag.mode)
      GET_DIAG(MODE := #statOtherInstruct.getDiag.mode, LADDR := #statDevDiagInternal.hwAddress[#statCntCyclGetDiag].hwtype5If, DIAG := #statOtherInstruct.getDiag.diagDataMode0, DETAIL :=, RET_VAL => #statOtherInstruct.getDiag.retVal, CNT_DIAG => #statOtherInstruct.getDiag.cntDiag)
   END_RUNG
   RUNG wire#w1
      Contact( #statOtherInstruct.getDiag.diagDataMode0.%X2 )
      Move(in := 2, out1 => #statOtherInstruct.getDiag.mode)
      GET_DIAG(MODE := #statOtherInstruct.getDiag.mode, LADDR := #statDevDiagInternal.hwAddress[#statCntCyclGetDiag].hwtype5If, DIAG := #statOtherInstruct.getDiag.diagDataMode2, DETAIL :=, RET_VAL => #statOtherInstruct.getDiag.retVal, CNT_DIAG => #statOtherInstruct.getDiag.cntDiag)
   END_RUNG
   RUNG wire#w1
      Contact( #statOtherInstruct.getDiag.diagDataMode0.%X1 )
      wire#w2
      Contact( #statOtherInstruct.getDiag.diagDataMode2.SubordinateIOState.%X4 )
      wire#w3
      I_Contact( #statOtherInstruct.getDiag.diagDataMode2.SubordinateIOState.%X15 )
      Contact( #statOtherInstruct.devStateMode4.state[#statCntCyclGetDiag] )
      wire#w4
      Coil( #interfaceDevDiag.devStateUser[#statCntCyclGetDiag].networkError )
   END_RUNG
   RUNG wire#w2
      Contact( #statOtherInstruct.getDiag.diagDataMode2.SubordinateIOState.%X5 )
   END_RUNG wire#w3
   RUNG wire#w4
      S_Coil( #statAlarm.deviceNetworkError )
   END_RUNG
   RUNG wire#w2
      Contact( #statOtherInstruct.getDiag.diagDataMode2.SubordinateIOState.%X2 )
      wire#w5
      Coil( #interfaceDevDiag.devStateUser[#statCntCyclGetDiag].maintenanceRequired )
   END_RUNG
   RUNG wire#w5
      S_Coil( #statAlarm.deviceMaintRequired )
   END_RUNG
   RUNG wire#w2
      Contact( #statOtherInstruct.getDiag.diagDataMode2.SubordinateIOState.%X3 )
      wire#w6
      Coil( #interfaceDevDiag.devStateUser[#statCntCyclGetDiag].maintenanceDemanded )
   END_RUNG
   RUNG wire#w6
      S_Coil( #statAlarm.deviceMaintDemanded )
   END_RUNG
   RUNG wire#w1
      { S7_Templates := "DestType := DInt" } Inc( #statCntCyclGetDiag )
   END_RUNG
   RUNG wire#w1
      { S7_Templates := "SrcType := DInt" } LT_Contact(in1 := #statDevDiagInternal.maxDevices, in2 := #statCntCyclGetDiag)
      Move(in := 1, out1 => #statCntCyclGetDiag)
   END_RUNG
   // the same network as SCL:
   IF #statBusy.getDiag THEN
       #statOtherInstruct.getDiag.mode := 0;
       #statOtherInstruct.getDiag.retVal := GET_DIAG(MODE := #statOtherInstruct.getDiag.mode,
                               LADDR := #statDevDiagInternal.hwAddress[#statCntCyclGetDiag].hwtype5If,
                               DIAG := #statOtherInstruct.getDiag.diagDataMode0,
                               CNT_DIAG => #statOtherInstruct.getDiag.cntDiag);
   END_IF;
   IF #statBusy.getDiag AND #statOtherInstruct.getDiag.diagDataMode0.%X2 THEN
       #statOtherInstruct.getDiag.mode := 2;
       #statOtherInstruct.getDiag.retVal := GET_DIAG(MODE := #statOtherInstruct.getDiag.mode,
                               LADDR := #statDevDiagInternal.hwAddress[#statCntCyclGetDiag].hwtype5If,
                               DIAG := #statOtherInstruct.getDiag.diagDataMode2,
                               CNT_DIAG => #statOtherInstruct.getDiag.cntDiag);
   END_IF;
   #_w1 := #statBusy.getDiag AND #statOtherInstruct.getDiag.diagDataMode0.%X1;
   #_w2 := #_w1 AND (#statOtherInstruct.getDiag.diagDataMode2.SubordinateIOState.%X4 OR #statOtherInstruct.getDiag.diagDataMode2.SubordinateIOState.%X5) AND NOT #statOtherInstruct.getDiag.diagDataMode2.SubordinateIOState.%X15 AND #statOtherInstruct.devStateMode4.state[#statCntCyclGetDiag];
   #interfaceDevDiag.devStateUser[#statCntCyclGetDiag].networkError := #_w1 AND (#statOtherInstruct.getDiag.diagDataMode2.SubordinateIOState.%X4 OR #statOtherInstruct.getDiag.diagDataMode2.SubordinateIOState.%X5) AND NOT #statOtherInstruct.getDiag.diagDataMode2.SubordinateIOState.%X15 AND #statOtherInstruct.devStateMode4.state[#statCntCyclGetDiag];
   IF #_w2 THEN #statAlarm.deviceNetworkError := TRUE; END_IF;
   #interfaceDevDiag.devStateUser[#statCntCyclGetDiag].maintenanceRequired := #_w1 AND #statOtherInstruct.getDiag.diagDataMode2.SubordinateIOState.%X2;
   IF #_w1 AND #statOtherInstruct.getDiag.diagDataMode2.SubordinateIOState.%X2 THEN
       #statAlarm.deviceMaintRequired := TRUE;
   END_IF;
   #interfaceDevDiag.devStateUser[#statCntCyclGetDiag].maintenanceDemanded := #_w1 AND #statOtherInstruct.getDiag.diagDataMode2.SubordinateIOState.%X3;
   IF #_w1 AND #statOtherInstruct.getDiag.diagDataMode2.SubordinateIOState.%X3 THEN
       #statAlarm.deviceMaintDemanded := TRUE;
   END_IF;
   IF #statBusy.getDiag THEN #statCntCyclGetDiag := #statCntCyclGetDiag + 1; END_IF;
   IF #statBusy.getDiag AND (#statDevDiagInternal.maxDevices < #statCntCyclGetDiag) THEN
       #statCntCyclGetDiag := 1;
   END_IF;
END_REGION

REGION Network 20: Read basic information / Lesen der Grundinformationen
   // Read the basic information only once via  "Get_IM_Data" / Einmaliges Lesen: GET_IM_DATA (I&M_0) der Grundinformationen
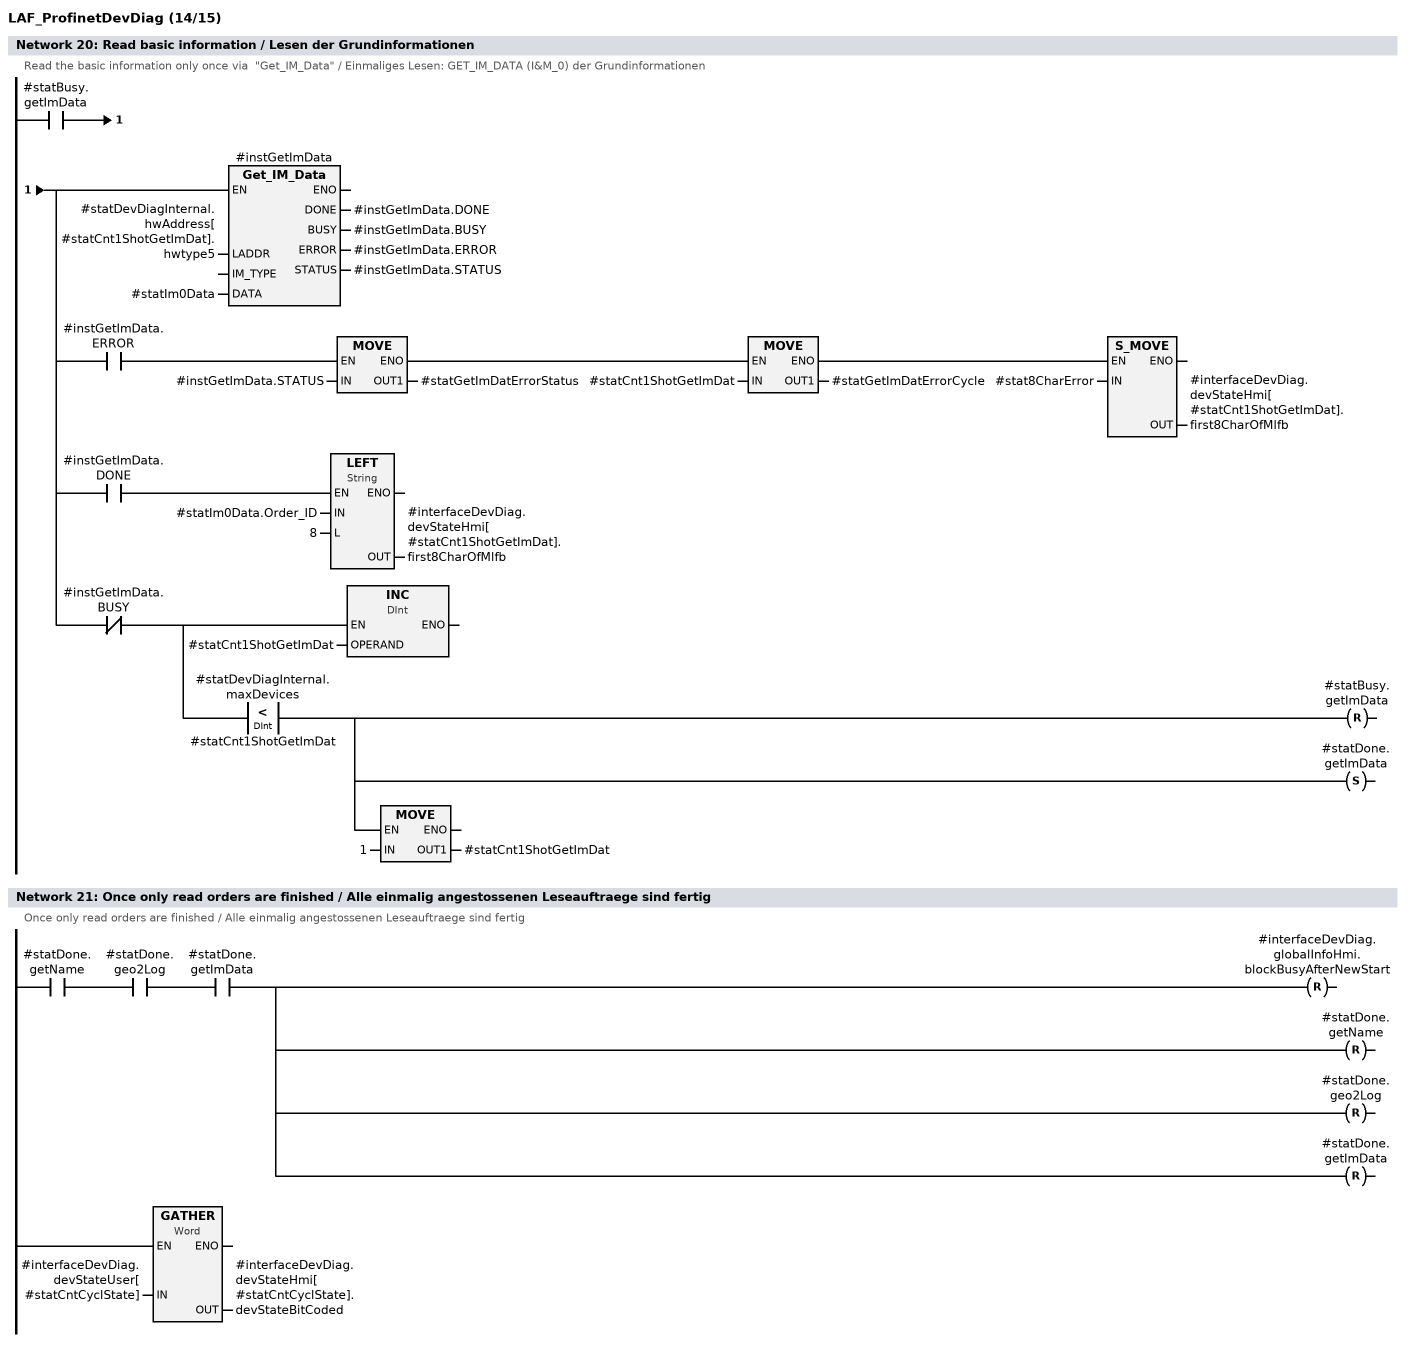
   RUNG wire#powerrail
      Contact( #statBusy.getImData )
      wire#w1
      #instGetImData.Get_IM_Data(LADDR := #statDevDiagInternal.hwAddress[#statCnt1ShotGetImDat].hwtype5, IM_TYPE :=, DATA := #statIm0Data, DONE => #instGetImData.DONE, BUSY => #instGetImData.BUSY, ERROR => #instGetImData.ERROR, STATUS => #instGetImData.STATUS)
   END_RUNG
   RUNG wire#w1
      Contact( #instGetImData.ERROR )
      Move(in := #instGetImData.STATUS, out1 => #statGetImDatErrorStatus)
      Move(in := #statCnt1ShotGetImDat, out1 => #statGetImDatErrorCycle)
      S_Move(in := #stat8CharError, out => #interfaceDevDiag.devStateHmi[#statCnt1ShotGetImDat].first8CharOfMlfb)
   END_RUNG
   RUNG wire#w1
      Contact( #instGetImData.DONE )
      { S7_Templates := "str_type := String" } LEFT(IN := #statIm0Data.Order_ID, L := 8, OUT => #interfaceDevDiag.devStateHmi[#statCnt1ShotGetImDat].first8CharOfMlfb)
   END_RUNG
   RUNG wire#w1
      I_Contact( #instGetImData.BUSY )
      wire#w2
      { S7_Templates := "DestType := DInt" } Inc( #statCnt1ShotGetImDat )
   END_RUNG
   RUNG wire#w2
      { S7_Templates := "SrcType := DInt" } LT_Contact(in1 := #statDevDiagInternal.maxDevices, in2 := #statCnt1ShotGetImDat)
      wire#w3
      R_Coil( #statBusy.getImData )
   END_RUNG
   RUNG wire#w3
      S_Coil( #statDone.getImData )
   END_RUNG
   RUNG wire#w3
      Move(in := 1, out1 => #statCnt1ShotGetImDat)
   END_RUNG
   // the same network as SCL:
   IF #statBusy.getImData THEN
       #instGetImData(LADDR := #statDevDiagInternal.hwAddress[#statCnt1ShotGetImDat].hwtype5,   // Get_IM_Data
                      DATA := #statIm0Data,
                      DONE => #instGetImData.DONE,
                      BUSY => #instGetImData.BUSY,
                      ERROR => #instGetImData.ERROR,
                      STATUS => #instGetImData.STATUS);
   END_IF;
   IF #statBusy.getImData AND #instGetImData.ERROR THEN
       #statGetImDatErrorStatus := #instGetImData.STATUS;
       #statGetImDatErrorCycle := #statCnt1ShotGetImDat;
       #interfaceDevDiag.devStateHmi[#statCnt1ShotGetImDat].first8CharOfMlfb := #stat8CharError;
   END_IF;
   IF #statBusy.getImData AND #instGetImData.DONE THEN
       LEFT(IN := #statIm0Data.Order_ID,
            L := 8,
            OUT => #interfaceDevDiag.devStateHmi[#statCnt1ShotGetImDat].first8CharOfMlfb);
   END_IF;
   #_w1 := #statBusy.getImData AND NOT #instGetImData.BUSY;
   IF #_w1 THEN #statCnt1ShotGetImDat := #statCnt1ShotGetImDat + 1; END_IF;
   IF #_w1 AND (#statDevDiagInternal.maxDevices < #statCnt1ShotGetImDat) THEN
       #statBusy.getImData := FALSE;
       #statDone.getImData := TRUE;
       #statCnt1ShotGetImDat := 1;
   END_IF;
END_REGION

REGION Network 21: Once only read orders are finished / Alle einmalig angestossenen Leseauftraege sind fertig
   // Once only read orders are finished / Alle einmalig angestossenen Leseauftraege sind fertig
   RUNG wire#powerrail
      Contact( #statDone.getName )
      Contact( #statDone.geo2Log )
      Contact( #statDone.getImData )
      wire#w1
      R_Coil( #interfaceDevDiag.globalInfoHmi.blockBusyAfterNewStart )
   END_RUNG
   RUNG wire#w1
      R_Coil( #statDone.getName )
   END_RUNG
   RUNG wire#w1
      R_Coil( #statDone.geo2Log )
   END_RUNG
   RUNG wire#w1
      R_Coil( #statDone.getImData )
   END_RUNG
   RUNG wire#powerrail
      { S7_Templates := "[dest_type := Word, src_type := Bool]" } GATHER(IN := #interfaceDevDiag.devStateUser[#statCntCyclState], OUT => #interfaceDevDiag.devStateHmi[#statCntCyclState].devStateBitCoded)
   END_RUNG
   // the same network as SCL:
   IF #statDone.getName AND #statDone.geo2Log AND #statDone.getImData THEN
       #interfaceDevDiag.globalInfoHmi.blockBusyAfterNewStart := FALSE;
   END_IF;
   #_w1 := #statDone.getName AND #statDone.geo2Log AND #statDone.getImData;
   IF #_w1 THEN
       #statDone.getName := FALSE;
       #statDone.geo2Log := FALSE;
       #statDone.getImData := FALSE;
   END_IF;
   GATHER(IN := #interfaceDevDiag.devStateUser[#statCntCyclState],
          OUT => #interfaceDevDiag.devStateHmi[#statCntCyclState].devStateBitCoded);
END_REGION

REGION Network 22: General Alarm / GENERAL Alarm
   // Transfer the alarms to outputs and generate summary alarm / Sammelalarm bilden / Alarme auf Qutput rangieren
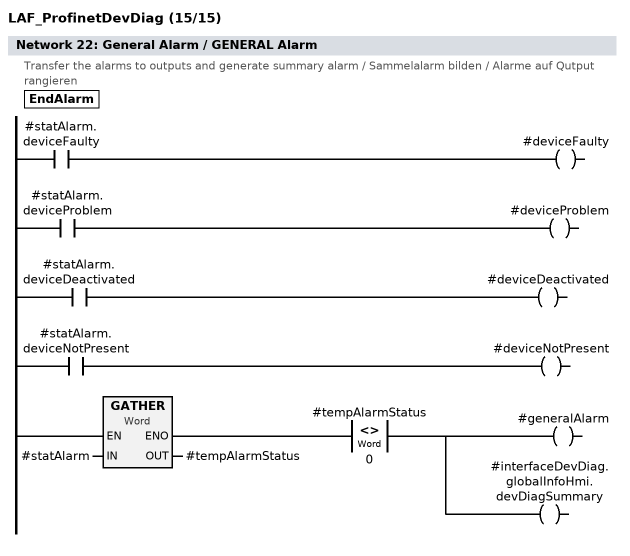
   Label( EndAlarm )
   RUNG wire#powerrail
      Contact( #statAlarm.deviceFaulty )
      Coil( #deviceFaulty )
   END_RUNG
   RUNG wire#powerrail
      Contact( #statAlarm.deviceProblem )
      Coil( #deviceProblem )
   END_RUNG
   RUNG wire#powerrail
      Contact( #statAlarm.deviceDeactivated )
      Coil( #deviceDeactivated )
   END_RUNG
   RUNG wire#powerrail
      Contact( #statAlarm.deviceNotPresent )
      Coil( #deviceNotPresent )
   END_RUNG
   RUNG wire#powerrail
      { S7_Templates := "[dest_type := Word, src_type := Bool]" } GATHER(IN := #statAlarm, OUT => #tempAlarmStatus)
      { S7_Templates := "SrcType := Word" } NE_Contact(in1 := #tempAlarmStatus, in2 := 0)
      wire#w1
      Coil( #generalAlarm )
   END_RUNG
   RUNG wire#w1
      Coil( #interfaceDevDiag.globalInfoHmi.devDiagSummary )
   END_RUNG
   // the same network as SCL:
   EndAlarm:
   #deviceFaulty := #statAlarm.deviceFaulty;
   #deviceProblem := #statAlarm.deviceProblem;
   #deviceDeactivated := #statAlarm.deviceDeactivated;
   #deviceNotPresent := #statAlarm.deviceNotPresent;
   GATHER(IN := #statAlarm, OUT => #tempAlarmStatus, ENO => #_w1);
   #generalAlarm := #_w1 AND (#tempAlarmStatus <> 0);
   #interfaceDevDiag.globalInfoHmi.devDiagSummary := #generalAlarm;
END_REGION
END_FUNCTION_BLOCK
